LIN {X 0,Y 413.536,Z 977.53,A -85,B 0,C 180,E1 16664.852,E2 16664.852} C_VEL
LIN {X 0,Y 413.201,Z 977.53,A -85,B 0,C 180,E1 16671.503,E2 16671.503} C_VEL
LIN {X 0,Y 412.887,Z 977.53,A -85,B 0,C 180,E1 16678.484,E2 16678.484} C_VEL
LIN {X 0,Y 412.713,Z 977.53,A -85,B 0,C 180,E1 16683.405,E2 16683.405} C_VEL
LIN {X 0,Y 412.557,Z 977.53,A -85,B 0,C 180,E1 16689.514,E2 16689.514} C_VEL
LIN {X 0,Y 412.491,Z 977.53,A -85,B 0,C 180,E1 16695.722,E2 16695.722} C_VEL
LIN {X 0,Y 412.588,Z 977.53,A -85,B 0,C 180,E1 16699.527,E2 16699.527} C_VEL
LIN {X 0,Y 434.551,Z 1034.787,A -85,B 0,C 180,E1 16702.862,E2 16702.862} C_VEL
LIN {X 0,Y 443.784,Z 1065.068,A -85,B 0,C 180,E1 16704.876,E2 16704.876} C_VEL
LIN {X 0,Y 438.617,Z 1105.248,A -85,B 0,C 180,E1 16707.191,E2 16707.191} C_VEL
LIN {X 0,Y 432.749,Z 1141.95,A -85,B 0,C 180,E1 16710.201,E2 16710.201} C_VEL
LIN {X 0,Y 427.169,Z 1174.246,A -85,B 0,C 180,E1 16713.808,E2 16713.808} C_VEL
LIN {X 0,Y 422.467,Z 1201.399,A -85,B 0,C 180,E1 16717.863,E2 16717.863} C_VEL
LIN {X 0,Y 418.685,Z 1224.945,A -85,B 0,C 180,E1 16722.615,E2 16722.615} C_VEL
LIN {X 0,Y 416.229,Z 1243.361,A -85,B 0,C 180,E1 16727.903,E2 16727.903} C_VEL
LIN {X 0,Y 415.214,Z 1254.307,A -85,B 0,C 180,E1 16732.648,E2 16732.648} C_VEL
LIN {X 0,Y 414.843,Z 1260.908,A -85,B 0,C 180,E1 16737.892,E2 16737.892} C_VEL
LIN {X 0,Y 415.006,Z 1262.266,A -85,B 0,C 180,E1 16742.077,E2 16742.077} C_VEL
LIN {X 0,Y 415.617,Z 1259.292,A -85,B 0,C 180,E1 16747.315,E2 16747.315} C_VEL
LIN {X 0,Y 417.308,Z 1251.014,A -85,B 0,C 180,E1 16752.567,E2 16752.567} C_VEL
LIN {X 0,Y 420.683,Z 1237.254,A -85,B 0,C 180,E1 16757.74,E2 16757.74} C_VEL
LIN {X 0,Y 426.06,Z 1217.939,A -85,B 0,C 180,E1 16762.692,E2 16762.692} C_VEL
LIN {X 0,Y 433.442,Z 1192.911,A -85,B 0,C 180,E1 16767.292,E2 16767.292} C_VEL
LIN {X 0,Y 442.539,Z 1161.806,A -85,B 0,C 180,E1 16771.457,E2 16771.457} C_VEL
LIN {X 0,Y 452.529,Z 1126.179,A -85,B 0,C 180,E1 16774.968,E2 16774.968} C_VEL
LIN {X 0,Y 462.553,Z 1087.333,A -85,B 0,C 180,E1 16777.725,E2 16777.725} C_VEL
LIN {X 0,Y 466.359,Z 1070.164,A -85,B 0,C 180,E1 16778.772,E2 16778.772} C_VEL
LIN {X 0,Y 465.511,Z 1057.108,A -85,B 0,C 180,E1 16780.595,E2 16780.595} C_VEL
LIN {X 0,Y 464.2,Z 1049.101,A -85,B 0,C 180,E1 16782.676,E2 16782.676} C_VEL
LIN {X 0,Y 464.109,Z 1045.742,A -85,B 0,C 180,E1 16784.686,E2 16784.686} C_VEL
LIN {X 0,Y 465.124,Z 1051.822,A -85,B 0,C 180,E1 16787.421,E2 16787.421} C_VEL
LIN {X 0,Y 465.932,Z 1056.52,A -85,B 0,C 180,E1 16788.389,E2 16788.389} C_VEL
LIN {X 0,Y 464.634,Z 1082.21,A -85,B 0,C 180,E1 16790.745,E2 16790.745} C_VEL
LIN {X 0,Y 453.94,Z 1125.674,A -85,B 0,C 180,E1 16793.081,E2 16793.081} C_VEL
LIN {X 0,Y 443.218,Z 1167.129,A -85,B 0,C 180,E1 16796.262,E2 16796.262} C_VEL
LIN {X 0,Y 434.228,Z 1201.819,A -85,B 0,C 180,E1 16799.903,E2 16799.903} C_VEL
LIN {X 0,Y 426.431,Z 1232.42,A -85,B 0,C 180,E1 16804.207,E2 16804.207} C_VEL
LIN {X 0,Y 420.735,Z 1257.224,A -85,B 0,C 180,E1 16808.901,E2 16808.901} C_VEL
LIN {X 0,Y 417.082,Z 1276.771,A -85,B 0,C 180,E1 16813.992,E2 16813.992} C_VEL
LIN {X 0,Y 415.427,Z 1289.933,A -85,B 0,C 180,E1 16818.97,E2 16818.97} C_VEL
LIN {X 0,Y 414.983,Z 1297.641,A -85,B 0,C 180,E1 16823.721,E2 16823.721} C_VEL
LIN {X 0,Y 414.942,Z 1300.55,A -85,B 0,C 180,E1 16827.917,E2 16827.917} C_VEL
LIN {X 0,Y 415.003,Z 1299.894,A -85,B 0,C 180,E1 16832.102,E2 16832.102} C_VEL
LIN {X 0,Y 415.091,Z 1293.746,A -85,B 0,C 180,E1 16837.35,E2 16837.35} C_VEL
LIN {X 0,Y 415.76,Z 1281.343,A -85,B 0,C 180,E1 16842.641,E2 16842.641} C_VEL
LIN {X 0,Y 416.754,Z 1270.596,A -85,B 0,C 180,E1 16845.839,E2 16845.839} C_VEL
LIN {X 0,Y 413.815,Z 1262.25,A -85,B 0,C 180,E1 16847.92,E2 16847.92} C_VEL
LIN {X 0,Y 411.157,Z 1253.033,A -85,B 0,C 180,E1 16849.975,E2 16849.975} C_VEL
LIN {X 0,Y 415.427,Z 1226.434,A -85,B 0,C 180,E1 16854.617,E2 16854.617} C_VEL
LIN {X 0,Y 423.644,Z 1186.586,A -85,B 0,C 180,E1 16860.06,E2 16860.06} C_VEL
LIN {X 0,Y 431.531,Z 1151.479,A -85,B 0,C 180,E1 16863.587,E2 16863.587} C_VEL
LIN {X 0,Y 439.938,Z 1112.289,A -85,B 0,C 180,E1 16866.462,E2 16866.462} C_VEL
LIN {X 0,Y 446.354,Z 1076.799,A -85,B 0,C 180,E1 16868.367,E2 16868.367} C_VEL
LIN {X 0,Y 443.694,Z 1053.032,A -85,B 0,C 180,E1 16870.272,E2 16870.272} C_VEL
LIN {X 0,Y 436.241,Z 1030.153,A -85,B 0,C 180,E1 16873.006,E2 16873.006} C_VEL
LIN {X 0,Y 428.199,Z 1013.282,A -85,B 0,C 180,E1 16876.073,E2 16876.073} C_VEL
LIN {X 0,Y 423.144,Z 1004.639,A -85,B 0,C 180,E1 16878.498,E2 16878.498} C_VEL
LIN {X 0,Y 420.285,Z 999.454,A -85,B 0,C 180,E1 16880.39,E2 16880.39} C_VEL
LIN {X 0,Y 416.589,Z 992.929,A -85,B 0,C 180,E1 16886.206,E2 16886.206} C_VEL
LIN {X 0,Y 419.779,Z 999.169,A -85,B 0,C 180,E1 16892.034,E2 16892.034} C_VEL
LIN {X 0,Y 426.481,Z 1011.08,A -85,B 0,C 180,E1 16896.342,E2 16896.342} C_VEL
LIN {X 0,Y 434.002,Z 1026.493,A -85,B 0,C 180,E1 16899.77,E2 16899.77} C_VEL
LIN {X 0,Y 441.381,Z 1046.678,A -85,B 0,C 180,E1 16902.741,E2 16902.741} C_VEL
LIN {X 0,Y 443.164,Z 1055.011,A -85,B 0,C 180,E1 16903.605,E2 16903.605} C_VEL
LIN {X 0,Y 435.927,Z 1100.938,A -85,B 0,C 180,E1 16905.934,E2 16905.934} C_VEL
LIN {X 0,Y 430.586,Z 1128.785,A -85,B 0,C 180,E1 16908.213,E2 16908.213} C_VEL
LIN {X 0,Y 424.859,Z 1152.118,A -85,B 0,C 180,E1 16911.039,E2 16911.039} C_VEL
LIN {X 0,Y 419.666,Z 1170.692,A -85,B 0,C 180,E1 16914.325,E2 16914.325} C_VEL
LIN {X 0,Y 414.89,Z 1185.812,A -85,B 0,C 180,E1 16918.446,E2 16918.446} C_VEL
LIN {X 0,Y 411.879,Z 1193.72,A -85,B 0,C 180,E1 16922.123,E2 16922.123} C_VEL
LIN {X 0,Y 409.732,Z 1197.42,A -85,B 0,C 180,E1 16926.384,E2 16926.384} C_VEL
LIN {X 0,Y 408.96,Z 1195.423,A -85,B 0,C 180,E1 16930.69,E2 16930.69} C_VEL
LIN {X 0,Y 409.267,Z 1187.552,A -85,B 0,C 180,E1 16935.034,E2 16935.034} C_VEL
LIN {X 0,Y 410.416,Z 1173.844,A -85,B 0,C 180,E1 16939.141,E2 16939.141} C_VEL
LIN {X 0,Y 412.34,Z 1154.397,A -85,B 0,C 180,E1 16942.905,E2 16942.905} C_VEL
LIN {X 0,Y 414.797,Z 1130.818,A -85,B 0,C 180,E1 16946.013,E2 16946.013} C_VEL
LIN {X 0,Y 417.4,Z 1103.039,A -85,B 0,C 180,E1 16948.484,E2 16948.484} C_VEL
LIN {X 0,Y 419.403,Z 1073.396,A -85,B 0,C 180,E1 16950.16,E2 16950.16} C_VEL
LIN {X 0,Y 420.294,Z 1032.093,A -85,B 0,C 180,E1 16951.546,E2 16951.546} C_VEL
LIN {X 0,Y 404.933,Z 977.53,A -85,B 0,C 180,E1 16954.16,E2 16954.16} C_VEL
LIN {X 0,Y 404.685,Z 977.53,A -85,B 0,C 180,E1 16961.493,E2 16961.493} C_VEL
LIN {X 0,Y 404.613,Z 977.53,A -85,B 0,C 180,E1 16968.519,E2 16968.519} C_VEL
LIN {X 0,Y 404.669,Z 977.53,A -85,B 0,C 180,E1 16975.817,E2 16975.817} C_VEL
LIN {X 0,Y 404.874,Z 977.53,A -85,B 0,C 180,E1 16980.876,E2 16980.876} C_VEL
LIN {X 0,Y 405.13,Z 977.53,A -85,B 0,C 180,E1 16985.695,E2 16985.695} C_VEL
LIN {X 0,Y 405.516,Z 977.53,A -85,B 0,C 180,E1 16992.596,E2 16992.596} C_VEL
LIN {X 0,Y 405.838,Z 977.53,A -85,B 0,C 180,E1 16999.231,E2 16999.231} C_VEL
LIN {X 0,Y 406.347,Z 977.53,A -85,B 0,C 180,E1 17005.713,E2 17005.713} C_VEL
LIN {X 0,Y 406.535,Z 977.53,A -85,B 0,C 180,E1 17012.126,E2 17012.126} C_VEL
LIN {X 0,Y 405.996,Z 977.53,A -85,B 0,C 180,E1 17018.576,E2 17018.576} C_VEL
LIN {X 0,Y 405.593,Z 977.53,A -85,B 0,C 180,E1 17025.15,E2 17025.15} C_VEL
LIN {X 0,Y 405.24,Z 977.53,A -85,B 0,C 180,E1 17031.947,E2 17031.947} C_VEL
LIN {X 0,Y 404.884,Z 977.53,A -85,B 0,C 180,E1 17039.101,E2 17039.101} C_VEL
LIN {X 0,Y 404.684,Z 977.53,A -85,B 0,C 180,E1 17044.521,E2 17044.521} C_VEL
LIN {X 0,Y 404.658,Z 977.53,A -85,B 0,C 180,E1 17051.488,E2 17051.488} C_VEL
LIN {X 0,Y 404.639,Z 977.53,A -85,B 0,C 180,E1 17058.914,E2 17058.914} C_VEL
LIN {X 0,Y 426.55,Z 1034.457,A -85,B 0,C 180,E1 17062.312,E2 17062.312} C_VEL
LIN {X 0,Y 436.463,Z 1066.891,A -85,B 0,C 180,E1 17064.525,E2 17064.525} C_VEL
LIN {X 0,Y 430.951,Z 1107.765,A -85,B 0,C 180,E1 17066.963,E2 17066.963} C_VEL
LIN {X 0,Y 424.975,Z 1144.124,A -85,B 0,C 180,E1 17070.042,E2 17070.042} C_VEL
LIN {X 0,Y 419.31,Z 1176.038,A -85,B 0,C 180,E1 17073.712,E2 17073.712} C_VEL
LIN {X 0,Y 414.384,Z 1203.666,A -85,B 0,C 180,E1 17077.974,E2 17077.974} C_VEL
LIN {X 0,Y 410.632,Z 1226.719,A -85,B 0,C 180,E1 17082.816,E2 17082.816} C_VEL
LIN {X 0,Y 408.424,Z 1243.246,A -85,B 0,C 180,E1 17087.669,E2 17087.669} C_VEL
LIN {X 0,Y 407.343,Z 1254.386,A -85,B 0,C 180,E1 17092.505,E2 17092.505} C_VEL
LIN {X 0,Y 406.977,Z 1261.213,A -85,B 0,C 180,E1 17097.851,E2 17097.851} C_VEL
LIN {X 0,Y 407.123,Z 1262.708,A -85,B 0,C 180,E1 17102.117,E2 17102.117} C_VEL
LIN {X 0,Y 407.801,Z 1259.921,A -85,B 0,C 180,E1 17107.456,E2 17107.456} C_VEL
LIN {X 0,Y 409.589,Z 1251.856,A -85,B 0,C 180,E1 17112.808,E2 17112.808} C_VEL
LIN {X 0,Y 413.286,Z 1238.13,A -85,B 0,C 180,E1 17118.139,E2 17118.139} C_VEL
LIN {X 0,Y 419.339,Z 1218.042,A -85,B 0,C 180,E1 17123.402,E2 17123.402} C_VEL
LIN {X 0,Y 427.658,Z 1191.664,A -85,B 0,C 180,E1 17128.268,E2 17128.268} C_VEL
LIN {X 0,Y 437.472,Z 1160.499,A -85,B 0,C 180,E1 17132.45,E2 17132.45} C_VEL
LIN {X 0,Y 448.599,Z 1123.62,A -85,B 0,C 180,E1 17136.048,E2 17136.048} C_VEL
LIN {X 0,Y 459.906,Z 1083.35,A -85,B 0,C 180,E1 17138.871,E2 17138.871} C_VEL
LIN {X 0,Y 462.155,Z 1073.258,A -85,B 0,C 180,E1 17139.544,E2 17139.544} C_VEL
LIN {X 0,Y 461.934,Z 1061.361,A -85,B 0,C 180,E1 17141.422,E2 17141.422} C_VEL
LIN {X 0,Y 461.315,Z 1054.684,A -85,B 0,C 180,E1 17143.741,E2 17143.741} C_VEL
LIN {X 0,Y 461.576,Z 1053.795,A -85,B 0,C 180,E1 17145.034,E2 17145.034} C_VEL
LIN {X 0,Y 462.268,Z 1059.274,A -85,B 0,C 180,E1 17147.264,E2 17147.264} C_VEL
LIN {X 0,Y 462.149,Z 1064.747,A -85,B 0,C 180,E1 17148.087,E2 17148.087} C_VEL
LIN {X 0,Y 459.961,Z 1085.959,A -85,B 0,C 180,E1 17150.036,E2 17150.036} C_VEL
LIN {X 0,Y 448.531,Z 1128.125,A -85,B 0,C 180,E1 17152.407,E2 17152.407} C_VEL
LIN {X 0,Y 436.938,Z 1169.453,A -85,B 0,C 180,E1 17155.711,E2 17155.711} C_VEL
LIN {X 0,Y 426.936,Z 1205.032,A -85,B 0,C 180,E1 17159.63,E2 17159.63} C_VEL
LIN {X 0,Y 418.917,Z 1234.622,A -85,B 0,C 180,E1 17163.998,E2 17163.998} C_VEL
LIN {X 0,Y 412.8,Z 1259.522,A -85,B 0,C 180,E1 17168.96,E2 17168.96} C_VEL
LIN {X 0,Y 409.067,Z 1278.74,A -85,B 0,C 180,E1 17174.304,E2 17174.304} C_VEL
LIN {X 0,Y 407.475,Z 1290.882,A -85,B 0,C 180,E1 17179.295,E2 17179.295} C_VEL
LIN {X 0,Y 407.093,Z 1297.34,A -85,B 0,C 180,E1 17183.599,E2 17183.599} C_VEL
LIN {X 0,Y 407.054,Z 1300.164,A -85,B 0,C 180,E1 17187.877,E2 17187.877} C_VEL
LIN {X 0,Y 407.111,Z 1299.389,A -85,B 0,C 180,E1 17192.143,E2 17192.143} C_VEL
LIN {X 0,Y 407.151,Z 1294.742,A -85,B 0,C 180,E1 17196.42,E2 17196.42} C_VEL
LIN {X 0,Y 407.568,Z 1284.889,A -85,B 0,C 180,E1 17201.266,E2 17201.266} C_VEL
LIN {X 0,Y 409.036,Z 1268.898,A -85,B 0,C 180,E1 17206.306,E2 17206.306} C_VEL
LIN {X 0,Y 411.157,Z 1253.033,A -85,B 0,C 180,E1 17209.975,E2 17209.975} C_VEL
LIN {X 0,Y 408.709,Z 1243.141,A -85,B 0,C 180,E1 17211.973,E2 17211.973} C_VEL
LIN {X 0,Y 406.726,Z 1232.323,A -85,B 0,C 180,E1 17213.894,E2 17213.894} C_VEL
LIN {X 0,Y 414.524,Z 1196.057,A -85,B 0,C 180,E1 17219.43,E2 17219.43} C_VEL
LIN {X 0,Y 422.708,Z 1161.586,A -85,B 0,C 180,E1 17223.303,E2 17223.303} C_VEL
LIN {X 0,Y 431.811,Z 1122.039,A -85,B 0,C 180,E1 17226.533,E2 17226.533} C_VEL
LIN {X 0,Y 440.546,Z 1079.46,A -85,B 0,C 180,E1 17228.968,E2 17228.968} C_VEL
LIN {X 0,Y 438.447,Z 1056.769,A -85,B 0,C 180,E1 17230.875,E2 17230.875} C_VEL
LIN {X 0,Y 431.79,Z 1034.922,A -85,B 0,C 180,E1 17233.622,E2 17233.622} C_VEL
LIN {X 0,Y 424.344,Z 1018.331,A -85,B 0,C 180,E1 17236.819,E2 17236.819} C_VEL
LIN {X 0,Y 418.261,Z 1007.062,A -85,B 0,C 180,E1 17240.432,E2 17240.432} C_VEL
LIN {X 0,Y 414.556,Z 1000.548,A -85,B 0,C 180,E1 17246.035,E2 17246.035} C_VEL
LIN {X 0,Y 415.519,Z 1004.822,A -85,B 0,C 180,E1 17250.297,E2 17250.297} C_VEL
LIN {X 0,Y 417.924,Z 1008.082,A -85,B 0,C 180,E1 17252.561,E2 17252.561} C_VEL
LIN {X 0,Y 424.057,Z 1019.723,A -85,B 0,C 180,E1 17256.566,E2 17256.566} C_VEL
LIN {X 0,Y 431.211,Z 1036.04,A -85,B 0,C 180,E1 17260.013,E2 17260.013} C_VEL
LIN {X 0,Y 437.52,Z 1056.068,A -85,B 0,C 180,E1 17262.818,E2 17262.818} C_VEL
LIN {X 0,Y 429.787,Z 1103.231,A -85,B 0,C 180,E1 17265.338,E2 17265.338} C_VEL
LIN {X 0,Y 424.151,Z 1130.371,A -85,B 0,C 180,E1 17267.639,E2 17267.639} C_VEL
LIN {X 0,Y 417.897,Z 1154.294,A -85,B 0,C 180,E1 17270.625,E2 17270.625} C_VEL
LIN {X 0,Y 412.226,Z 1173.211,A -85,B 0,C 180,E1 17274.129,E2 17274.129} C_VEL
LIN {X 0,Y 407.693,Z 1186.506,A -85,B 0,C 180,E1 17277.885,E2 17277.885} C_VEL
LIN {X 0,Y 404.055,Z 1195.396,A -85,B 0,C 180,E1 17282.164,E2 17282.164} C_VEL
LIN {X 0,Y 401.849,Z 1198.507,A -85,B 0,C 180,E1 17286.51,E2 17286.51} C_VEL
LIN {X 0,Y 401.121,Z 1196.049,A -85,B 0,C 180,E1 17290.902,E2 17290.902} C_VEL
LIN {X 0,Y 401.451,Z 1187.613,A -85,B 0,C 180,E1 17295.334,E2 17295.334} C_VEL
LIN {X 0,Y 402.68,Z 1173.379,A -85,B 0,C 180,E1 17299.523,E2 17299.523} C_VEL
LIN {X 0,Y 404.655,Z 1153.91,A -85,B 0,C 180,E1 17303.244,E2 17303.244} C_VEL
LIN {X 0,Y 407.234,Z 1129.906,A -85,B 0,C 180,E1 17306.384,E2 17306.384} C_VEL
LIN {X 0,Y 409.884,Z 1102.27,A -85,B 0,C 180,E1 17308.834,E2 17308.834} C_VEL
LIN {X 0,Y 411.856,Z 1071.439,A -85,B 0,C 180,E1 17310.558,E2 17310.558} C_VEL
LIN {X 0,Y 412.97,Z 1034.333,A -85,B 0,C 180,E1 17311.814,E2 17311.814} C_VEL
LIN {X 0,Y 396.984,Z 977.53,A -85,B 0,C 180,E1 17314.608,E2 17314.608} C_VEL
LIN {X 0,Y 396.738,Z 977.53,A -85,B 0,C 180,E1 17320.502,E2 17320.502} C_VEL
LIN {X 0,Y 396.628,Z 977.53,A -85,B 0,C 180,E1 17326.557,E2 17326.557} C_VEL
LIN {X 0,Y 396.697,Z 977.53,A -85,B 0,C 180,E1 17333.352,E2 17333.352} C_VEL
LIN {X 0,Y 396.933,Z 977.53,A -85,B 0,C 180,E1 17340.235,E2 17340.235} C_VEL
LIN {X 0,Y 397.284,Z 977.53,A -85,B 0,C 180,E1 17347.568,E2 17347.568} C_VEL
LIN {X 0,Y 397.651,Z 977.53,A -85,B 0,C 180,E1 17354.519,E2 17354.519} C_VEL
LIN {X 0,Y 398.124,Z 977.53,A -85,B 0,C 180,E1 17361.776,E2 17361.776} C_VEL
LIN {X 0,Y 398.591,Z 977.53,A -85,B 0,C 180,E1 17367.811,E2 17367.811} C_VEL
LIN {X 0,Y 398.623,Z 977.53,A -85,B 0,C 180,E1 17372.168,E2 17372.168} C_VEL
LIN {X 0,Y 398.066,Z 977.53,A -85,B 0,C 180,E1 17378.748,E2 17378.748} C_VEL
LIN {X 0,Y 397.64,Z 977.53,A -85,B 0,C 180,E1 17385.46,E2 17385.46} C_VEL
LIN {X 0,Y 397.255,Z 977.53,A -85,B 0,C 180,E1 17392.411,E2 17392.411} C_VEL
LIN {X 0,Y 396.938,Z 977.53,A -85,B 0,C 180,E1 17399.741,E2 17399.741} C_VEL
LIN {X 0,Y 396.726,Z 977.53,A -85,B 0,C 180,E1 17406.654,E2 17406.654} C_VEL
LIN {X 0,Y 396.66,Z 977.53,A -85,B 0,C 180,E1 17413.448,E2 17413.448} C_VEL
LIN {X 0,Y 396.705,Z 977.53,A -85,B 0,C 180,E1 17418.264,E2 17418.264} C_VEL
LIN {X 0,Y 419.101,Z 1035.699,A -85,B 0,C 180,E1 17421.852,E2 17421.852} C_VEL
LIN {X 0,Y 429.116,Z 1068.588,A -85,B 0,C 180,E1 17424.155,E2 17424.155} C_VEL
LIN {X 0,Y 423.515,Z 1108.732,A -85,B 0,C 180,E1 17426.614,E2 17426.614} C_VEL
LIN {X 0,Y 417.45,Z 1144.782,A -85,B 0,C 180,E1 17429.726,E2 17429.726} C_VEL
LIN {X 0,Y 411.631,Z 1176.792,A -85,B 0,C 180,E1 17433.478,E2 17433.478} C_VEL
LIN {X 0,Y 406.586,Z 1204.37,A -85,B 0,C 180,E1 17437.817,E2 17437.817} C_VEL
LIN {X 0,Y 402.761,Z 1227.315,A -85,B 0,C 180,E1 17442.742,E2 17442.742} C_VEL
LIN {X 0,Y 400.434,Z 1244.556,A -85,B 0,C 180,E1 17447.973,E2 17447.973} C_VEL
LIN {X 0,Y 399.488,Z 1254.42,A -85,B 0,C 180,E1 17452.356,E2 17452.356} C_VEL
LIN {X 0,Y 399.078,Z 1261.475,A -85,B 0,C 180,E1 17457.809,E2 17457.809} C_VEL
LIN {X 0,Y 399.234,Z 1263.156,A -85,B 0,C 180,E1 17462.159,E2 17462.159} C_VEL
LIN {X 0,Y 399.974,Z 1260.569,A -85,B 0,C 180,E1 17467.603,E2 17467.603} C_VEL
LIN {X 0,Y 401.881,Z 1252.733,A -85,B 0,C 180,E1 17473.058,E2 17473.058} C_VEL
LIN {X 0,Y 405.841,Z 1239.276,A -85,B 0,C 180,E1 17478.485,E2 17478.485} C_VEL
LIN {X 0,Y 412.219,Z 1219.565,A -85,B 0,C 180,E1 17483.831,E2 17483.831} C_VEL
LIN {X 0,Y 420.995,Z 1193.848,A -85,B 0,C 180,E1 17488.756,E2 17488.756} C_VEL
LIN {X 0,Y 431.625,Z 1162.505,A -85,B 0,C 180,E1 17493.095,E2 17493.095} C_VEL
LIN {X 0,Y 443.394,Z 1126.739,A -85,B 0,C 180,E1 17496.708,E2 17496.708} C_VEL
LIN {X 0,Y 455.543,Z 1087.183,A -85,B 0,C 180,E1 17499.59,E2 17499.59} C_VEL
LIN {X 0,Y 458.267,Z 1076.739,A -85,B 0,C 180,E1 17500.305,E2 17500.305} C_VEL
LIN {X 0,Y 458.594,Z 1066.761,A -85,B 0,C 180,E1 17502.065,E2 17502.065} C_VEL
LIN {X 0,Y 458.613,Z 1061.998,A -85,B 0,C 180,E1 17503.91,E2 17503.91} C_VEL
LIN {X 0,Y 458.836,Z 1061.482,A -85,B 0,C 180,E1 17505.063,E2 17505.063} C_VEL
LIN {X 0,Y 459.199,Z 1065.972,A -85,B 0,C 180,E1 17506.909,E2 17506.909} C_VEL
LIN {X 0,Y 456.734,Z 1084.393,A -85,B 0,C 180,E1 17508.934,E2 17508.934} C_VEL
LIN {X 0,Y 441.705,Z 1136.16,A -85,B 0,C 180,E1 17512.106,E2 17512.106} C_VEL
LIN {X 0,Y 429.188,Z 1176.718,A -85,B 0,C 180,E1 17515.617,E2 17515.617} C_VEL
LIN {X 0,Y 418.299,Z 1212.873,A -85,B 0,C 180,E1 17519.97,E2 17519.97} C_VEL
LIN {X 0,Y 410.135,Z 1241.628,A -85,B 0,C 180,E1 17524.676,E2 17524.676} C_VEL
LIN {X 0,Y 404.633,Z 1263.027,A -85,B 0,C 180,E1 17529.361,E2 17529.361} C_VEL
LIN {X 0,Y 400.982,Z 1280.599,A -85,B 0,C 180,E1 17534.672,E2 17534.672} C_VEL
LIN {X 0,Y 399.507,Z 1292.048,A -85,B 0,C 180,E1 17539.837,E2 17539.837} C_VEL
LIN {X 0,Y 399.195,Z 1297.048,A -85,B 0,C 180,E1 17543.472,E2 17543.472} C_VEL
LIN {X 0,Y 399.156,Z 1299.775,A -85,B 0,C 180,E1 17547.835,E2 17547.835} C_VEL
LIN {X 0,Y 399.22,Z 1298.841,A -85,B 0,C 180,E1 17552.185,E2 17552.185} C_VEL
LIN {X 0,Y 399.264,Z 1294.081,A -85,B 0,C 180,E1 17556.548,E2 17556.548} C_VEL
LIN {X 0,Y 399.715,Z 1284.023,A -85,B 0,C 180,E1 17561.49,E2 17561.49} C_VEL
LIN {X 0,Y 401.192,Z 1268.398,A -85,B 0,C 180,E1 17566.466,E2 17566.466} C_VEL
LIN {X 0,Y 404.142,Z 1247.252,A -85,B 0,C 180,E1 17571.248,E2 17571.248} C_VEL
LIN {X 0,Y 406.726,Z 1232.323,A -85,B 0,C 180,E1 17573.894,E2 17573.894} C_VEL
LIN {X 0,Y 405.15,Z 1221.758,A -85,B 0,C 180,E1 17575.852,E2 17575.852} C_VEL
LIN {X 0,Y 403.783,Z 1211.089,A -85,B 0,C 180,E1 17577.819,E2 17577.819} C_VEL
LIN {X 0,Y 411.821,Z 1179.033,A -85,B 0,C 180,E1 17582.112,E2 17582.112} C_VEL
LIN {X 0,Y 421.33,Z 1141.248,A -85,B 0,C 180,E1 17585.793,E2 17585.793} C_VEL
LIN {X 0,Y 430.998,Z 1100.356,A -85,B 0,C 180,E1 17588.624,E2 17588.624} C_VEL
LIN {X 0,Y 434.777,Z 1080.838,A -85,B 0,C 180,E1 17589.697,E2 17589.697} C_VEL
LIN {X 0,Y 433.109,Z 1059.718,A -85,B 0,C 180,E1 17591.582,E2 17591.582} C_VEL
LIN {X 0,Y 426.991,Z 1038.703,A -85,B 0,C 180,E1 17594.426,E2 17594.426} C_VEL
LIN {X 0,Y 420.286,Z 1023.051,A -85,B 0,C 180,E1 17597.698,E2 17597.698} C_VEL
LIN {X 0,Y 415.391,Z 1014.15,A -85,B 0,C 180,E1 17600.949,E2 17600.949} C_VEL
LIN {X 0,Y 412.407,Z 1008.203,A -85,B 0,C 180,E1 17605.695,E2 17605.695} C_VEL
LIN {X 0,Y 412.319,Z 1010.467,A -85,B 0,C 180,E1 17608.7,E2 17608.7} C_VEL
LIN {X 0,Y 415.089,Z 1015.364,A -85,B 0,C 180,E1 17612.357,E2 17612.357} C_VEL
LIN {X 0,Y 420.765,Z 1026.999,A -85,B 0,C 180,E1 17616.403,E2 17616.403} C_VEL
LIN {X 0,Y 427.441,Z 1043.484,A -85,B 0,C 180,E1 17619.884,E2 17619.884} C_VEL
LIN {X 0,Y 432.021,Z 1060.552,A -85,B 0,C 180,E1 17622.244,E2 17622.244} C_VEL
LIN {X 0,Y 424.074,Z 1103.904,A -85,B 0,C 180,E1 17624.605,E2 17624.605} C_VEL
LIN {X 0,Y 417.817,Z 1132.19,A -85,B 0,C 180,E1 17627.049,E2 17627.049} C_VEL
LIN {X 0,Y 410.962,Z 1156.535,A -85,B 0,C 180,E1 17630.198,E2 17630.198} C_VEL
LIN {X 0,Y 405.257,Z 1174.219,A -85,B 0,C 180,E1 17633.576,E2 17633.576} C_VEL
LIN {X 0,Y 399.957,Z 1188.755,A -85,B 0,C 180,E1 17637.845,E2 17637.845} C_VEL
LIN {X 0,Y 396.233,Z 1196.962,A -85,B 0,C 180,E1 17642.207,E2 17642.207} C_VEL
LIN {X 0,Y 393.97,Z 1199.598,A -85,B 0,C 180,E1 17646.641,E2 17646.641} C_VEL
LIN {X 0,Y 393.258,Z 1196.591,A -85,B 0,C 180,E1 17651.123,E2 17651.123} C_VEL
LIN {X 0,Y 393.685,Z 1187.339,A -85,B 0,C 180,E1 17655.76,E2 17655.76} C_VEL
LIN {X 0,Y 395.011,Z 1172.824,A -85,B 0,C 180,E1 17659.906,E2 17659.906} C_VEL
LIN {X 0,Y 397.105,Z 1153.015,A -85,B 0,C 180,E1 17663.657,E2 17663.657} C_VEL
LIN {X 0,Y 399.795,Z 1127.631,A -85,B 0,C 180,E1 17666.914,E2 17666.914} C_VEL
LIN {X 0,Y 402.455,Z 1099.688,A -85,B 0,C 180,E1 17669.319,E2 17669.319} C_VEL
LIN {X 0,Y 404.451,Z 1068.492,A -85,B 0,C 180,E1 17670.995,E2 17670.995} C_VEL
LIN {X 0,Y 405.272,Z 1035.045,A -85,B 0,C 180,E1 17672.148,E2 17672.148} C_VEL
LIN {X 0,Y 389.001,Z 977.53,A -85,B 0,C 180,E1 17675.096,E2 17675.096} C_VEL
LIN {X 0,Y 388.68,Z 977.53,A -85,B 0,C 180,E1 17682.193,E2 17682.193} C_VEL
LIN {X 0,Y 388.635,Z 977.53,A -85,B 0,C 180,E1 17688.471,E2 17688.471} C_VEL
LIN {X 0,Y 388.8,Z 977.53,A -85,B 0,C 180,E1 17694.946,E2 17694.946} C_VEL
LIN {X 0,Y 389.054,Z 977.53,A -85,B 0,C 180,E1 17702.125,E2 17702.125} C_VEL
LIN {X 0,Y 389.463,Z 977.53,A -85,B 0,C 180,E1 17709.492,E2 17709.492} C_VEL
LIN {X 0,Y 389.851,Z 977.53,A -85,B 0,C 180,E1 17716.503,E2 17716.503} C_VEL
LIN {X 0,Y 390.369,Z 977.53,A -85,B 0,C 180,E1 17723.302,E2 17723.302} C_VEL
LIN {X 0,Y 390.881,Z 977.53,A -85,B 0,C 180,E1 17729.99,E2 17729.99} C_VEL
LIN {X 0,Y 390.332,Z 977.53,A -85,B 0,C 180,E1 17736.677,E2 17736.677} C_VEL
LIN {X 0,Y 389.838,Z 977.53,A -85,B 0,C 180,E1 17743.617,E2 17743.617} C_VEL
LIN {X 0,Y 389.406,Z 977.53,A -85,B 0,C 180,E1 17750.923,E2 17750.923} C_VEL
LIN {X 0,Y 389.054,Z 977.53,A -85,B 0,C 180,E1 17757.852,E2 17757.852} C_VEL
LIN {X 0,Y 388.864,Z 977.53,A -85,B 0,C 180,E1 17765.068,E2 17765.068} C_VEL
LIN {X 0,Y 388.687,Z 977.53,A -85,B 0,C 180,E1 17772.193,E2 17772.193} C_VEL
LIN {X 0,Y 388.845,Z 978.262,A -85,B 0,C 180,E1 17777.674,E2 17777.674} C_VEL
LIN {X 0,Y 410.325,Z 1033.448,A -85,B 0,C 180,E1 17781.138,E2 17781.138} C_VEL
LIN {X 0,Y 421.734,Z 1070.249,A -85,B 0,C 180,E1 17783.782,E2 17783.782} C_VEL
LIN {X 0,Y 416.111,Z 1109.544,A -85,B 0,C 180,E1 17786.253,E2 17786.253} C_VEL
LIN {X 0,Y 409.883,Z 1145.668,A -85,B 0,C 180,E1 17789.435,E2 17789.435} C_VEL
LIN {X 0,Y 403.97,Z 1177.456,A -85,B 0,C 180,E1 17793.235,E2 17793.235} C_VEL
LIN {X 0,Y 398.788,Z 1205.002,A -85,B 0,C 180,E1 17797.654,E2 17797.654} C_VEL
LIN {X 0,Y 394.922,Z 1227.672,A -85,B 0,C 180,E1 17802.613,E2 17802.613} C_VEL
LIN {X 0,Y 392.609,Z 1244.393,A -85,B 0,C 180,E1 17807.73,E2 17807.73} C_VEL
LIN {X 0,Y 391.618,Z 1254.437,A -85,B 0,C 180,E1 17812.202,E2 17812.202} C_VEL
LIN {X 0,Y 391.189,Z 1261.717,A -85,B 0,C 180,E1 17817.765,E2 17817.765} C_VEL
LIN {X 0,Y 391.361,Z 1263.605,A -85,B 0,C 180,E1 17822.203,E2 17822.203} C_VEL
LIN {X 0,Y 391.867,Z 1262.108,A -85,B 0,C 180,E1 17826.645,E2 17826.645} C_VEL
LIN {X 0,Y 393.671,Z 1255.563,A -85,B 0,C 180,E1 17832.204,E2 17832.204} C_VEL
LIN {X 0,Y 397.312,Z 1243.592,A -85,B 0,C 180,E1 17837.746,E2 17837.746} C_VEL
LIN {X 0,Y 403.819,Z 1224.829,A -85,B 0,C 180,E1 17843.408,E2 17843.408} C_VEL
LIN {X 0,Y 412.763,Z 1200.513,A -85,B 0,C 180,E1 17848.484,E2 17848.484} C_VEL
LIN {X 0,Y 423.128,Z 1172.44,A -85,B 0,C 180,E1 17852.774,E2 17852.774} C_VEL
LIN {X 0,Y 435.535,Z 1137.932,A -85,B 0,C 180,E1 17856.66,E2 17856.66} C_VEL
LIN {X 0,Y 449.097,Z 1098.521,A -85,B 0,C 180,E1 17859.848,E2 17859.848} C_VEL
LIN {X 0,Y 454.543,Z 1081.55,A -85,B 0,C 180,E1 17860.939,E2 17860.939} C_VEL
LIN {X 0,Y 455.425,Z 1073.391,A -85,B 0,C 180,E1 17862.426,E2 17862.426} C_VEL
LIN {X 0,Y 455.796,Z 1069.201,A -85,B 0,C 180,E1 17864.252,E2 17864.252} C_VEL
LIN {X 0,Y 456.008,Z 1071.424,A -85,B 0,C 180,E1 17866.175,E2 17866.175} C_VEL
LIN {X 0,Y 455.611,Z 1074.544,A -85,B 0,C 180,E1 17866.763,E2 17866.763} C_VEL
LIN {X 0,Y 452.214,Z 1091.112,A -85,B 0,C 180,E1 17868.416,E2 17868.416} C_VEL
LIN {X 0,Y 438.117,Z 1134.084,A -85,B 0,C 180,E1 17871.033,E2 17871.033} C_VEL
LIN {X 0,Y 424.153,Z 1175.777,A -85,B 0,C 180,E1 17874.681,E2 17874.681} C_VEL
LIN {X 0,Y 412.454,Z 1211.637,A -85,B 0,C 180,E1 17879.059,E2 17879.059} C_VEL
LIN {X 0,Y 403.687,Z 1239.752,A -85,B 0,C 180,E1 17883.685,E2 17883.685} C_VEL
LIN {X 0,Y 397.393,Z 1262.1,A -85,B 0,C 180,E1 17888.626,E2 17888.626} C_VEL
LIN {X 0,Y 393.521,Z 1279.282,A -85,B 0,C 180,E1 17893.858,E2 17893.858} C_VEL
LIN {X 0,Y 391.645,Z 1291.668,A -85,B 0,C 180,E1 17899.504,E2 17899.504} C_VEL
LIN {X 0,Y 391.315,Z 1296.763,A -85,B 0,C 180,E1 17903.339,E2 17903.339} C_VEL
LIN {X 0,Y 391.258,Z 1299.389,A -85,B 0,C 180,E1 17907.791,E2 17907.791} C_VEL
LIN {X 0,Y 391.357,Z 1298.286,A -85,B 0,C 180,E1 17912.229,E2 17912.229} C_VEL
LIN {X 0,Y 391.381,Z 1293.402,A -85,B 0,C 180,E1 17916.68,E2 17916.68} C_VEL
LIN {X 0,Y 391.895,Z 1283.119,A -85,B 0,C 180,E1 17921.722,E2 17921.722} C_VEL
LIN {X 0,Y 393.456,Z 1267.225,A -85,B 0,C 180,E1 17926.799,E2 17926.799} C_VEL
LIN {X 0,Y 396.471,Z 1246.163,A -85,B 0,C 180,E1 17931.594,E2 17931.594} C_VEL
LIN {X 0,Y 403.783,Z 1211.089,A -85,B 0,C 180,E1 17937.819,E2 17937.819} C_VEL
LIN {X 0,Y 402.993,Z 1200.026,A -85,B 0,C 180,E1 17939.749,E2 17939.749} C_VEL
LIN {X 0,Y 402.754,Z 1188.376,A -85,B 0,C 180,E1 17941.614,E2 17941.614} C_VEL
LIN {X 0,Y 412.441,Z 1152.501,A -85,B 0,C 180,E1 17945.528,E2 17945.528} C_VEL
LIN {X 0,Y 422.357,Z 1113.696,A -85,B 0,C 180,E1 17948.573,E2 17948.573} C_VEL
LIN {X 0,Y 429.164,Z 1082.342,A -85,B 0,C 180,E1 17950.447,E2 17950.447} C_VEL
LIN {X 0,Y 428.047,Z 1063.831,A -85,B 0,C 180,E1 17952.178,E2 17952.178} C_VEL
LIN {X 0,Y 422.672,Z 1043.689,A -85,B 0,C 180,E1 17955.047,E2 17955.047} C_VEL
LIN {X 0,Y 416.915,Z 1029.278,A -85,B 0,C 180,E1 17958.23,E2 17958.23} C_VEL
LIN {X 0,Y 412.722,Z 1021.415,A -85,B 0,C 180,E1 17961.25,E2 17961.25} C_VEL
LIN {X 0,Y 410.04,Z 1015.71,A -85,B 0,C 180,E1 17966.359,E2 17966.359} C_VEL
LIN {X 0,Y 412.069,Z 1022.185,A -85,B 0,C 180,E1 17971.97,E2 17971.97} C_VEL
LIN {X 0,Y 416.807,Z 1032.693,A -85,B 0,C 180,E1 17975.828,E2 17975.828} C_VEL
LIN {X 0,Y 422.958,Z 1049.005,A -85,B 0,C 180,E1 17979.421,E2 17979.421} C_VEL
LIN {X 0,Y 426.643,Z 1063.348,A -85,B 0,C 180,E1 17981.529,E2 17981.529} C_VEL
LIN {X 0,Y 418.201,Z 1106.168,A -85,B 0,C 180,E1 17983.95,E2 17983.95} C_VEL
LIN {X 0,Y 411.522,Z 1134.031,A -85,B 0,C 180,E1 17986.441,E2 17986.441} C_VEL
LIN {X 0,Y 404.629,Z 1157.175,A -85,B 0,C 180,E1 17989.498,E2 17989.498} C_VEL
LIN {X 0,Y 398.1,Z 1176.08,A -85,B 0,C 180,E1 17993.185,E2 17993.185} C_VEL
LIN {X 0,Y 392.821,Z 1189.539,A -85,B 0,C 180,E1 17997.252,E2 17997.252} C_VEL
LIN {X 0,Y 389.178,Z 1197.16,A -85,B 0,C 180,E1 18001.131,E2 18001.131} C_VEL
LIN {X 0,Y 387.069,Z 1200.283,A -85,B 0,C 180,E1 18004.506,E2 18004.506} C_VEL
LIN {X 0,Y 385.552,Z 1199.561,A -85,B 0,C 180,E1 18009.06,E2 18009.06} C_VEL
LIN {X 0,Y 385.504,Z 1193.161,A -85,B 0,C 180,E1 18013.656,E2 18013.656} C_VEL
LIN {X 0,Y 386.353,Z 1181.233,A -85,B 0,C 180,E1 18018.005,E2 18018.005} C_VEL
LIN {X 0,Y 388.138,Z 1163.661,A -85,B 0,C 180,E1 18022.085,E2 18022.085} C_VEL
LIN {X 0,Y 390.711,Z 1141.76,A -85,B 0,C 180,E1 18025.533,E2 18025.533} C_VEL
LIN {X 0,Y 393.333,Z 1116.179,A -85,B 0,C 180,E1 18028.329,E2 18028.329} C_VEL
LIN {X 0,Y 395.858,Z 1087.075,A -85,B 0,C 180,E1 18030.427,E2 18030.427} C_VEL
LIN {X 0,Y 397.658,Z 1052.431,A -85,B 0,C 180,E1 18031.887,E2 18031.887} C_VEL
LIN {X 0,Y 397.638,Z 1036.142,A -85,B 0,C 180,E1 18032.473,E2 18032.473} C_VEL
LIN {X 0,Y 381.039,Z 977.53,A -85,B 0,C 180,E1 18035.537,E2 18035.537} C_VEL
LIN {X 0,Y 380.724,Z 977.53,A -85,B 0,C 180,E1 18042.594,E2 18042.594} C_VEL
LIN {X 0,Y 380.661,Z 977.53,A -85,B 0,C 180,E1 18049.157,E2 18049.157} C_VEL
LIN {X 0,Y 380.921,Z 977.53,A -85,B 0,C 180,E1 18056.672,E2 18056.672} C_VEL
LIN {X 0,Y 381.235,Z 977.53,A -85,B 0,C 180,E1 18064.062,E2 18064.062} C_VEL
LIN {X 0,Y 381.627,Z 977.53,A -85,B 0,C 180,E1 18071.468,E2 18071.468} C_VEL
LIN {X 0,Y 382.037,Z 977.53,A -85,B 0,C 180,E1 18078.551,E2 18078.551} C_VEL
LIN {X 0,Y 382.614,Z 977.53,A -85,B 0,C 180,E1 18085.447,E2 18085.447} C_VEL
LIN {X 0,Y 382.978,Z 977.53,A -85,B 0,C 180,E1 18089.989,E2 18089.989} C_VEL
LIN {X 0,Y 382.399,Z 977.53,A -85,B 0,C 180,E1 18096.817,E2 18096.817} C_VEL
LIN {X 0,Y 381.93,Z 977.53,A -85,B 0,C 180,E1 18103.76,E2 18103.76} C_VEL
LIN {X 0,Y 381.517,Z 977.53,A -85,B 0,C 180,E1 18110.932,E2 18110.932} C_VEL
LIN {X 0,Y 381.05,Z 977.53,A -85,B 0,C 180,E1 18118.49,E2 18118.49} C_VEL
LIN {X 0,Y 380.941,Z 977.53,A -85,B 0,C 180,E1 18123.827,E2 18123.827} C_VEL
LIN {X 0,Y 380.733,Z 977.53,A -85,B 0,C 180,E1 18130.855,E2 18130.855} C_VEL
LIN {X 0,Y 380.866,Z 977.913,A -85,B 0,C 180,E1 18136.982,E2 18136.982} C_VEL
LIN {X 0,Y 402.828,Z 1034.577,A -85,B 0,C 180,E1 18140.648,E2 18140.648} C_VEL
LIN {X 0,Y 414.384,Z 1071.969,A -85,B 0,C 180,E1 18143.411,E2 18143.411} C_VEL
LIN {X 0,Y 408.408,Z 1112.007,A -85,B 0,C 180,E1 18146.01,E2 18146.01} C_VEL
LIN {X 0,Y 401.918,Z 1148.964,A -85,B 0,C 180,E1 18149.392,E2 18149.392} C_VEL
LIN {X 0,Y 395.71,Z 1181.37,A -85,B 0,C 180,E1 18153.453,E2 18153.453} C_VEL
LIN {X 0,Y 390.408,Z 1208.841,A -85,B 0,C 180,E1 18158.129,E2 18158.129} C_VEL
LIN {X 0,Y 386.848,Z 1229.558,A -85,B 0,C 180,E1 18162.901,E2 18162.901} C_VEL
LIN {X 0,Y 384.62,Z 1245.661,A -85,B 0,C 180,E1 18168.048,E2 18168.048} C_VEL
LIN {X 0,Y 383.546,Z 1256.406,A -85,B 0,C 180,E1 18173.178,E2 18173.178} C_VEL
LIN {X 0,Y 383.291,Z 1261.949,A -85,B 0,C 180,E1 18177.718,E2 18177.718} C_VEL
LIN {X 0,Y 383.473,Z 1264.057,A -85,B 0,C 180,E1 18182.248,E2 18182.248} C_VEL
LIN {X 0,Y 384.04,Z 1262.716,A -85,B 0,C 180,E1 18186.781,E2 18186.781} C_VEL
LIN {X 0,Y 385.947,Z 1256.423,A -85,B 0,C 180,E1 18192.452,E2 18192.452} C_VEL
LIN {X 0,Y 389.85,Z 1244.753,A -85,B 0,C 180,E1 18198.097,E2 18198.097} C_VEL
LIN {X 0,Y 396.684,Z 1226.571,A -85,B 0,C 180,E1 18203.813,E2 18203.813} C_VEL
LIN {X 0,Y 406.129,Z 1202.786,A -85,B 0,C 180,E1 18208.993,E2 18208.993} C_VEL
LIN {X 0,Y 417.564,Z 1174.131,A -85,B 0,C 180,E1 18213.515,E2 18213.515} C_VEL
LIN {X 0,Y 431.217,Z 1139.264,A -85,B 0,C 180,E1 18217.538,E2 18217.538} C_VEL
LIN {X 0,Y 445.487,Z 1101.494,A -85,B 0,C 180,E1 18220.664,E2 18220.664} C_VEL
LIN {X 0,Y 451.252,Z 1085.433,A -85,B 0,C 180,E1 18221.735,E2 18221.735} C_VEL
LIN {X 0,Y 452.462,Z 1078.353,A -85,B 0,C 180,E1 18223.33,E2 18223.33} C_VEL
LIN {X 0,Y 452.802,Z 1076.825,A -85,B 0,C 180,E1 18224.622,E2 18224.622} C_VEL
LIN {X 0,Y 452.95,Z 1078.428,A -85,B 0,C 180,E1 18225.918,E2 18225.918} C_VEL
LIN {X 0,Y 448.965,Z 1093.664,A -85,B 0,C 180,E1 18227.558,E2 18227.558} C_VEL
LIN {X 0,Y 433.698,Z 1135.792,A -85,B 0,C 180,E1 18230.201,E2 18230.201} C_VEL
LIN {X 0,Y 418.494,Z 1177.466,A -85,B 0,C 180,E1 18233.97,E2 18233.97} C_VEL
LIN {X 0,Y 405.842,Z 1213.176,A -85,B 0,C 180,E1 18238.498,E2 18238.498} C_VEL
LIN {X 0,Y 396.723,Z 1240.263,A -85,B 0,C 180,E1 18243.112,E2 18243.112} C_VEL
LIN {X 0,Y 389.898,Z 1262.72,A -85,B 0,C 180,E1 18248.256,E2 18248.256} C_VEL
LIN {X 0,Y 385.525,Z 1280.709,A -85,B 0,C 180,E1 18254.041,E2 18254.041} C_VEL
LIN {X 0,Y 383.704,Z 1292.487,A -85,B 0,C 180,E1 18259.889,E2 18259.889} C_VEL
LIN {X 0,Y 383.34,Z 1298.189,A -85,B 0,C 180,E1 18265.476,E2 18265.476} C_VEL
LIN {X 0,Y 383.586,Z 1298.844,A -85,B 0,C 180,E1 18270.011,E2 18270.011} C_VEL
LIN {X 0,Y 383.537,Z 1294.336,A -85,B 0,C 180,E1 18275.679,E2 18275.679} C_VEL
LIN {X 0,Y 383.826,Z 1285.179,A -85,B 0,C 180,E1 18280.761,E2 18280.761} C_VEL
LIN {X 0,Y 385.303,Z 1269.177,A -85,B 0,C 180,E1 18286.283,E2 18286.283} C_VEL
LIN {X 0,Y 388.446,Z 1247.485,A -85,B 0,C 180,E1 18291.462,E2 18291.462} C_VEL
LIN {X 0,Y 396.603,Z 1211.42,A -85,B 0,C 180,E1 18298.308,E2 18298.308} C_VEL
LIN {X 0,Y 402.754,Z 1188.376,A -85,B 0,C 180,E1 18301.614,E2 18301.614} C_VEL
LIN {X 0,Y 402.89,Z 1176.339,A -85,B 0,C 180,E1 18303.427,E2 18303.427} C_VEL
LIN {X 0,Y 403.218,Z 1163.741,A -85,B 0,C 180,E1 18305.151,E2 18305.151} C_VEL
LIN {X 0,Y 414.118,Z 1124.223,A -85,B 0,C 180,E1 18308.645,E2 18308.645} C_VEL
LIN {X 0,Y 423.714,Z 1083.801,A -85,B 0,C 180,E1 18311.233,E2 18311.233} C_VEL
LIN {X 0,Y 423.042,Z 1067.916,A -85,B 0,C 180,E1 18312.803,E2 18312.803} C_VEL
LIN {X 0,Y 418.604,Z 1049.336,A -85,B 0,C 180,E1 18315.566,E2 18315.566} C_VEL
LIN {X 0,Y 413.478,Z 1035.468,A -85,B 0,C 180,E1 18318.753,E2 18318.753} C_VEL
LIN {X 0,Y 410.477,Z 1029.081,A -85,B 0,C 180,E1 18321.155,E2 18321.155} C_VEL
LIN {X 0,Y 407.65,Z 1023.248,A -85,B 0,C 180,E1 18326.136,E2 18326.136} C_VEL
LIN {X 0,Y 409.271,Z 1029.8,A -85,B 0,C 180,E1 18331.93,E2 18331.93} C_VEL
LIN {X 0,Y 413.402,Z 1039.732,A -85,B 0,C 180,E1 18335.616,E2 18335.616} C_VEL
LIN {X 0,Y 418.935,Z 1056.034,A -85,B 0,C 180,E1 18339.214,E2 18339.214} C_VEL
LIN {X 0,Y 421.306,Z 1066.749,A -85,B 0,C 180,E1 18340.809,E2 18340.809} C_VEL
LIN {X 0,Y 412.541,Z 1108.095,A -85,B 0,C 180,E1 18343.239,E2 18343.239} C_VEL
LIN {X 0,Y 405.348,Z 1136.067,A -85,B 0,C 180,E1 18345.817,E2 18345.817} C_VEL
LIN {X 0,Y 397.235,Z 1161.18,A -85,B 0,C 180,E1 18349.3,E2 18349.3} C_VEL
LIN {X 0,Y 390.127,Z 1180.083,A -85,B 0,C 180,E1 18353.325,E2 18353.325} C_VEL
LIN {X 0,Y 384.472,Z 1193.026,A -85,B 0,C 180,E1 18357.758,E2 18357.758} C_VEL
LIN {X 0,Y 380.557,Z 1200.072,A -85,B 0,C 180,E1 18362.298,E2 18362.298} C_VEL
LIN {X 0,Y 378.21,Z 1201.592,A -85,B 0,C 180,E1 18366.919,E2 18366.919} C_VEL
LIN {X 0,Y 377.543,Z 1197.567,A -85,B 0,C 180,E1 18371.592,E2 18371.592} C_VEL
LIN {X 0,Y 378.059,Z 1187.474,A -85,B 0,C 180,E1 18376.309,E2 18376.309} C_VEL
LIN {X 0,Y 379.622,Z 1171.687,A -85,B 0,C 180,E1 18380.679,E2 18380.679} C_VEL
LIN {X 0,Y 381.984,Z 1150.524,A -85,B 0,C 180,E1 18384.572,E2 18384.572} C_VEL
LIN {X 0,Y 384.768,Z 1125.541,A -85,B 0,C 180,E1 18387.716,E2 18387.716} C_VEL
LIN {X 0,Y 387.559,Z 1096.76,A -85,B 0,C 180,E1 18390.158,E2 18390.158} C_VEL
LIN {X 0,Y 389.577,Z 1065.006,A -85,B 0,C 180,E1 18391.793,E2 18391.793} C_VEL
LIN {X 0,Y 390.056,Z 1037.279,A -85,B 0,C 180,E1 18392.806,E2 18392.806} C_VEL
LIN {X 0,Y 373.063,Z 977.53,A -85,B 0,C 180,E1 18396.084,E2 18396.084} C_VEL
LIN {X 0,Y 372.794,Z 977.53,A -85,B 0,C 180,E1 18403.725,E2 18403.725} C_VEL
LIN {X 0,Y 372.766,Z 977.53,A -85,B 0,C 180,E1 18410.582,E2 18410.582} C_VEL
LIN {X 0,Y 373.044,Z 977.53,A -85,B 0,C 180,E1 18418.56,E2 18418.56} C_VEL
LIN {X 0,Y 373.442,Z 977.53,A -85,B 0,C 180,E1 18426.05,E2 18426.05} C_VEL
LIN {X 0,Y 373.822,Z 977.53,A -85,B 0,C 180,E1 18433.505,E2 18433.505} C_VEL
LIN {X 0,Y 374.286,Z 977.53,A -85,B 0,C 180,E1 18440.67,E2 18440.67} C_VEL
LIN {X 0,Y 374.862,Z 977.53,A -85,B 0,C 180,E1 18447.673,E2 18447.673} C_VEL
LIN {X 0,Y 374.887,Z 977.53,A -85,B 0,C 180,E1 18452.306,E2 18452.306} C_VEL
LIN {X 0,Y 374.263,Z 977.53,A -85,B 0,C 180,E1 18459.309,E2 18459.309} C_VEL
LIN {X 0,Y 373.795,Z 977.53,A -85,B 0,C 180,E1 18466.473,E2 18466.473} C_VEL
LIN {X 0,Y 373.402,Z 977.53,A -85,B 0,C 180,E1 18473.929,E2 18473.929} C_VEL
LIN {X 0,Y 373.038,Z 977.53,A -85,B 0,C 180,E1 18481.861,E2 18481.861} C_VEL
LIN {X 0,Y 372.827,Z 977.53,A -85,B 0,C 180,E1 18489.429,E2 18489.429} C_VEL
LIN {X 0,Y 372.921,Z 977.93,A -85,B 0,C 180,E1 18496.294,E2 18496.294} C_VEL
LIN {X 0,Y 395.04,Z 1034.8,A -85,B 0,C 180,E1 18500.082,E2 18500.082} C_VEL
LIN {X 0,Y 407.052,Z 1073.3,A -85,B 0,C 180,E1 18503.016,E2 18503.016} C_VEL
LIN {X 0,Y 401.125,Z 1112.09,A -85,B 0,C 180,E1 18505.582,E2 18505.582} C_VEL
LIN {X 0,Y 394.593,Z 1148.222,A -85,B 0,C 180,E1 18508.921,E2 18508.921} C_VEL
LIN {X 0,Y 388.181,Z 1181.216,A -85,B 0,C 180,E1 18513.093,E2 18513.093} C_VEL
LIN {X 0,Y 382.751,Z 1208.576,A -85,B 0,C 180,E1 18517.802,E2 18517.802} C_VEL
LIN {X 0,Y 378.972,Z 1230.093,A -85,B 0,C 180,E1 18522.835,E2 18522.835} C_VEL
LIN {X 0,Y 376.801,Z 1245.453,A -85,B 0,C 180,E1 18527.796,E2 18527.796} C_VEL
LIN {X 0,Y 375.67,Z 1256.46,A -85,B 0,C 180,E1 18533.034,E2 18533.034} C_VEL
LIN {X 0,Y 375.395,Z 1262.172,A -85,B 0,C 180,E1 18537.67,E2 18537.67} C_VEL
LIN {X 0,Y 375.599,Z 1264.499,A -85,B 0,C 180,E1 18542.295,E2 18542.295} C_VEL
LIN {X 0,Y 376.221,Z 1263.334,A -85,B 0,C 180,E1 18546.922,E2 18546.922} C_VEL
LIN {X 0,Y 378.233,Z 1257.318,A -85,B 0,C 180,E1 18552.711,E2 18552.711} C_VEL
LIN {X 0,Y 382.426,Z 1245.966,A -85,B 0,C 180,E1 18558.461,E2 18558.461} C_VEL
LIN {X 0,Y 389.371,Z 1228.805,A -85,B 0,C 180,E1 18564.112,E2 18564.112} C_VEL
LIN {X 0,Y 399.567,Z 1205.191,A -85,B 0,C 180,E1 18569.516,E2 18569.516} C_VEL
LIN {X 0,Y 412.435,Z 1175.343,A -85,B 0,C 180,E1 18574.37,E2 18574.37} C_VEL
LIN {X 0,Y 427.315,Z 1140.573,A -85,B 0,C 180,E1 18578.465,E2 18578.465} C_VEL
LIN {X 0,Y 442.841,Z 1103.117,A -85,B 0,C 180,E1 18581.612,E2 18581.612} C_VEL
LIN {X 0,Y 448.175,Z 1089.695,A -85,B 0,C 180,E1 18582.522,E2 18582.522} C_VEL
LIN {X 0,Y 449.298,Z 1085.196,A -85,B 0,C 180,E1 18583.715,E2 18583.715} C_VEL
LIN {X 0,Y 449.699,Z 1084.391,A -85,B 0,C 180,E1 18585.013,E2 18585.013} C_VEL
LIN {X 0,Y 449.105,Z 1086.72,A -85,B 0,C 180,E1 18585.629,E2 18585.629} C_VEL
LIN {X 0,Y 445.97,Z 1096.475,A -85,B 0,C 180,E1 18586.683,E2 18586.683} C_VEL
LIN {X 0,Y 429.736,Z 1137.318,A -85,B 0,C 180,E1 18589.312,E2 18589.312} C_VEL
LIN {X 0,Y 412.938,Z 1179.344,A -85,B 0,C 180,E1 18593.244,E2 18593.244} C_VEL
LIN {X 0,Y 399.922,Z 1213.155,A -85,B 0,C 180,E1 18597.656,E2 18597.656} C_VEL
LIN {X 0,Y 389.415,Z 1242.146,A -85,B 0,C 180,E1 18602.774,E2 18602.774} C_VEL
LIN {X 0,Y 382.026,Z 1264.83,A -85,B 0,C 180,E1 18608.269,E2 18608.269} C_VEL
LIN {X 0,Y 377.463,Z 1282.392,A -85,B 0,C 180,E1 18614.374,E2 18614.374} C_VEL
LIN {X 0,Y 375.857,Z 1292.178,A -85,B 0,C 180,E1 18619.559,E2 18619.559} C_VEL
LIN {X 0,Y 375.443,Z 1297.865,A -85,B 0,C 180,E1 18625.381,E2 18625.381} C_VEL
LIN {X 0,Y 375.699,Z 1298.33,A -85,B 0,C 180,E1 18630.011,E2 18630.011} C_VEL
LIN {X 0,Y 375.589,Z 1295.036,A -85,B 0,C 180,E1 18634.639,E2 18634.639} C_VEL
LIN {X 0,Y 375.842,Z 1286.643,A -85,B 0,C 180,E1 18639.877,E2 18639.877} C_VEL
LIN {X 0,Y 376.996,Z 1273.127,A -85,B 0,C 180,E1 18645.062,E2 18645.062} C_VEL
LIN {X 0,Y 379.677,Z 1253.24,A -85,B 0,C 180,E1 18650.34,E2 18650.34} C_VEL
LIN {X 0,Y 387.654,Z 1218.395,A -85,B 0,C 180,E1 18657.668,E2 18657.668} C_VEL
LIN {X 0,Y 396.388,Z 1187.568,A -85,B 0,C 180,E1 18662.368,E2 18662.368} C_VEL
LIN {X 0,Y 403.218,Z 1163.741,A -85,B 0,C 180,E1 18665.151,E2 18665.151} C_VEL
LIN {X 0,Y 403.88,Z 1150.806,A -85,B 0,C 180,E1 18666.843,E2 18666.843} C_VEL
LIN {X 0,Y 404.409,Z 1139.231,A -85,B 0,C 180,E1 18668.267,E2 18668.267} C_VEL
LIN {X 0,Y 404.882,Z 1137.407,A -85,B 0,C 180,E1 18668.426,E2 18668.426} C_VEL
LIN {X 0,Y 416.82,Z 1094.375,A -85,B 0,C 180,E1 18671.428,E2 18671.428} C_VEL
LIN {X 0,Y 418.413,Z 1085.704,A -85,B 0,C 180,E1 18672.007,E2 18672.007} C_VEL
LIN {X 0,Y 417.934,Z 1071.113,A -85,B 0,C 180,E1 18673.554,E2 18673.554} C_VEL
LIN {X 0,Y 414.129,Z 1053.82,A -85,B 0,C 180,E1 18676.316,E2 18676.316} C_VEL
LIN {X 0,Y 410.006,Z 1041.688,A -85,B 0,C 180,E1 18679.292,E2 18679.292} C_VEL
LIN {X 0,Y 407.729,Z 1036.443,A -85,B 0,C 180,E1 18681.316,E2 18681.316} C_VEL
LIN {X 0,Y 405.078,Z 1031.013,A -85,B 0,C 180,E1 18685.891,E2 18685.891} C_VEL
LIN {X 0,Y 405.807,Z 1035.551,A -85,B 0,C 180,E1 18690.982,E2 18690.982} C_VEL
LIN {X 0,Y 409.519,Z 1045.603,A -85,B 0,C 180,E1 18695.066,E2 18695.066} C_VEL
LIN {X 0,Y 414.242,Z 1060.594,A -85,B 0,C 180,E1 18698.562,E2 18698.562} C_VEL
LIN {X 0,Y 416,Z 1070.629,A -85,B 0,C 180,E1 18700.09,E2 18700.09} C_VEL
LIN {X 0,Y 406.876,Z 1110.661,A -85,B 0,C 180,E1 18702.545,E2 18702.545} C_VEL
LIN {X 0,Y 399.212,Z 1138.159,A -85,B 0,C 180,E1 18705.173,E2 18705.173} C_VEL
LIN {X 0,Y 391.018,Z 1161.971,A -85,B 0,C 180,E1 18708.562,E2 18708.562} C_VEL
LIN {X 0,Y 383.836,Z 1179.865,A -85,B 0,C 180,E1 18712.361,E2 18712.361} C_VEL
LIN {X 0,Y 378.051,Z 1192.676,A -85,B 0,C 180,E1 18716.57,E2 18716.57} C_VEL
LIN {X 0,Y 373.531,Z 1200.454,A -85,B 0,C 180,E1 18721.179,E2 18721.179} C_VEL
LIN {X 0,Y 371.326,Z 1202.725,A -85,B 0,C 180,E1 18724.698,E2 18724.698} C_VEL
LIN {X 0,Y 369.831,Z 1200.957,A -85,B 0,C 180,E1 18729.448,E2 18729.448} C_VEL
LIN {X 0,Y 369.864,Z 1193.419,A -85,B 0,C 180,E1 18734.245,E2 18734.245} C_VEL
LIN {X 0,Y 370.89,Z 1180.375,A -85,B 0,C 180,E1 18738.783,E2 18738.783} C_VEL
LIN {X 0,Y 372.95,Z 1161.379,A -85,B 0,C 180,E1 18743.035,E2 18743.035} C_VEL
LIN {X 0,Y 375.719,Z 1138.317,A -85,B 0,C 180,E1 18746.539,E2 18746.539} C_VEL
LIN {X 0,Y 378.567,Z 1111.219,A -85,B 0,C 180,E1 18749.377,E2 18749.377} C_VEL
LIN {X 0,Y 381.121,Z 1080.853,A -85,B 0,C 180,E1 18751.428,E2 18751.428} C_VEL
LIN {X 0,Y 382.67,Z 1039.271,A -85,B 0,C 180,E1 18753.105,E2 18753.105} C_VEL
LIN {X 0,Y 365.108,Z 977.53,A -85,B 0,C 180,E1 18756.557,E2 18756.557} C_VEL
LIN {X 0,Y 364.857,Z 977.53,A -85,B 0,C 180,E1 18761.66,E2 18761.66} C_VEL
LIN {X 0,Y 364.804,Z 977.53,A -85,B 0,C 180,E1 18768.406,E2 18768.406} C_VEL
LIN {X 0,Y 364.907,Z 977.53,A -85,B 0,C 180,E1 18774.441,E2 18774.441} C_VEL
LIN {X 0,Y 365.213,Z 977.53,A -85,B 0,C 180,E1 18780.631,E2 18780.631} C_VEL
LIN {X 0,Y 365.577,Z 977.53,A -85,B 0,C 180,E1 18788.085,E2 18788.085} C_VEL
LIN {X 0,Y 366.021,Z 977.53,A -85,B 0,C 180,E1 18795.606,E2 18795.606} C_VEL
LIN {X 0,Y 366.589,Z 977.53,A -85,B 0,C 180,E1 18802.866,E2 18802.866} C_VEL
LIN {X 0,Y 367.17,Z 977.53,A -85,B 0,C 180,E1 18809.989,E2 18809.989} C_VEL
LIN {X 0,Y 366.549,Z 977.53,A -85,B 0,C 180,E1 18817.113,E2 18817.113} C_VEL
LIN {X 0,Y 366.014,Z 977.53,A -85,B 0,C 180,E1 18824.371,E2 18824.371} C_VEL
LIN {X 0,Y 365.564,Z 977.53,A -85,B 0,C 180,E1 18831.892,E2 18831.892} C_VEL
LIN {X 0,Y 365.157,Z 977.53,A -85,B 0,C 180,E1 18839.852,E2 18839.852} C_VEL
LIN {X 0,Y 364.955,Z 977.53,A -85,B 0,C 180,E1 18845.526,E2 18845.526} C_VEL
LIN {X 0,Y 364.846,Z 977.53,A -85,B 0,C 180,E1 18851.629,E2 18851.629} C_VEL
LIN {X 0,Y 364.959,Z 977.53,A -85,B 0,C 180,E1 18855.551,E2 18855.551} C_VEL
LIN {X 0,Y 387.487,Z 1035.851,A -85,B 0,C 180,E1 18859.565,E2 18859.565} C_VEL
LIN {X 0,Y 399.559,Z 1073.863,A -85,B 0,C 180,E1 18862.55,E2 18862.55} C_VEL
LIN {X 0,Y 393.598,Z 1113.677,A -85,B 0,C 180,E1 18865.266,E2 18865.266} C_VEL
LIN {X 0,Y 386.865,Z 1150.037,A -85,B 0,C 180,E1 18868.722,E2 18868.722} C_VEL
LIN {X 0,Y 380.223,Z 1182.999,A -85,B 0,C 180,E1 18873.028,E2 18873.028} C_VEL
LIN {X 0,Y 374.875,Z 1209.495,A -85,B 0,C 180,E1 18877.717,E2 18877.717} C_VEL
LIN {X 0,Y 371.094,Z 1230.589,A -85,B 0,C 180,E1 18882.765,E2 18882.765} C_VEL
LIN {X 0,Y 368.815,Z 1246.676,A -85,B 0,C 180,E1 18888.13,E2 18888.13} C_VEL
LIN {X 0,Y 367.797,Z 1256.488,A -85,B 0,C 180,E1 18892.884,E2 18892.884} C_VEL
LIN {X 0,Y 367.498,Z 1262.385,A -85,B 0,C 180,E1 18897.62,E2 18897.62} C_VEL
LIN {X 0,Y 367.707,Z 1264.889,A -85,B 0,C 180,E1 18902.345,E2 18902.345} C_VEL
LIN {X 0,Y 368.396,Z 1263.969,A -85,B 0,C 180,E1 18907.07,E2 18907.07} C_VEL
LIN {X 0,Y 370.548,Z 1258.24,A -85,B 0,C 180,E1 18912.979,E2 18912.979} C_VEL
LIN {X 0,Y 375.019,Z 1247.239,A -85,B 0,C 180,E1 18918.839,E2 18918.839} C_VEL
LIN {X 0,Y 382.413,Z 1230.408,A -85,B 0,C 180,E1 18924.622,E2 18924.622} C_VEL
LIN {X 0,Y 393.678,Z 1206.31,A -85,B 0,C 180,E1 18930.321,E2 18930.321} C_VEL
LIN {X 0,Y 408.218,Z 1175.277,A -85,B 0,C 180,E1 18935.456,E2 18935.456} C_VEL
LIN {X 0,Y 424.597,Z 1140.194,A -85,B 0,C 180,E1 18939.603,E2 18939.603} C_VEL
LIN {X 0,Y 441.917,Z 1102.167,A -85,B 0,C 180,E1 18942.767,E2 18942.767} C_VEL
LIN {X 0,Y 445.375,Z 1094.158,A -85,B 0,C 180,E1 18943.338,E2 18943.338} C_VEL
LIN {X 0,Y 446.237,Z 1091.872,A -85,B 0,C 180,E1 18944.526,E2 18944.526} C_VEL
LIN {X 0,Y 446,Z 1092.776,A -85,B 0,C 180,E1 18945.047,E2 18945.047} C_VEL
LIN {X 0,Y 443.222,Z 1099.884,A -85,B 0,C 180,E1 18945.815,E2 18945.815} C_VEL
LIN {X 0,Y 425.128,Z 1141.314,A -85,B 0,C 180,E1 18948.589,E2 18948.589} C_VEL
LIN {X 0,Y 407.044,Z 1182.539,A -85,B 0,C 180,E1 18952.622,E2 18952.622} C_VEL
LIN {X 0,Y 392.129,Z 1218.28,A -85,B 0,C 180,E1 18957.578,E2 18957.578} C_VEL
LIN {X 0,Y 381.439,Z 1245.807,A -85,B 0,C 180,E1 18962.829,E2 18962.829} C_VEL
LIN {X 0,Y 374.384,Z 1265.947,A -85,B 0,C 180,E1 18968.026,E2 18968.026} C_VEL
LIN {X 0,Y 369.643,Z 1282.943,A -85,B 0,C 180,E1 18974.254,E2 18974.254} C_VEL
LIN {X 0,Y 367.885,Z 1293.537,A -85,B 0,C 180,E1 18980.528,E2 18980.528} C_VEL
LIN {X 0,Y 367.538,Z 1297.54,A -85,B 0,C 180,E1 18985.281,E2 18985.281} C_VEL
LIN {X 0,Y 367.813,Z 1297.808,A -85,B 0,C 180,E1 18990.011,E2 18990.011} C_VEL
LIN {X 0,Y 367.708,Z 1294.379,A -85,B 0,C 180,E1 18994.738,E2 18994.738} C_VEL
LIN {X 0,Y 367.986,Z 1285.743,A -85,B 0,C 180,E1 19000.09,E2 19000.09} C_VEL
LIN {X 0,Y 369.183,Z 1271.939,A -85,B 0,C 180,E1 19005.389,E2 19005.389} C_VEL
LIN {X 0,Y 372.093,Z 1251.461,A -85,B 0,C 180,E1 19010.839,E2 19010.839} C_VEL
LIN {X 0,Y 378.732,Z 1224.484,A -85,B 0,C 180,E1 19017.083,E2 19017.083} C_VEL
LIN {X 0,Y 387.862,Z 1194.077,A -85,B 0,C 180,E1 19022.172,E2 19022.172} C_VEL
LIN {X 0,Y 397.944,Z 1161.169,A -85,B 0,C 180,E1 19026.184,E2 19026.184} C_VEL
LIN {X 0,Y 404.882,Z 1137.407,A -85,B 0,C 180,E1 19028.426,E2 19028.426} C_VEL
LIN {X 0,Y 406.35,Z 1123.589,A -85,B 0,C 180,E1 19029.94,E2 19029.94} C_VEL
LIN {X 0,Y 407.863,Z 1109.439,A -85,B 0,C 180,E1 19031.372,E2 19031.372} C_VEL
LIN {X 0,Y 413.243,Z 1088.327,A -85,B 0,C 180,E1 19032.746,E2 19032.746} C_VEL
LIN {X 0,Y 413.113,Z 1075.37,A -85,B 0,C 180,E1 19034.193,E2 19034.193} C_VEL
LIN {X 0,Y 410.08,Z 1059.337,A -85,B 0,C 180,E1 19036.879,E2 19036.879} C_VEL
LIN {X 0,Y 406.927,Z 1048.894,A -85,B 0,C 180,E1 19039.481,E2 19039.481} C_VEL
LIN {X 0,Y 404.364,Z 1043.218,A -85,B 0,C 180,E1 19041.915,E2 19041.915} C_VEL
LIN {X 0,Y 402.4,Z 1038.528,A -85,B 0,C 180,E1 19045.955,E2 19045.955} C_VEL
LIN {X 0,Y 402.81,Z 1042.695,A -85,B 0,C 180,E1 19050.745,E2 19050.745} C_VEL
LIN {X 0,Y 405.521,Z 1051.088,A -85,B 0,C 180,E1 19054.353,E2 19054.353} C_VEL
LIN {X 0,Y 409.413,Z 1064.391,A -85,B 0,C 180,E1 19057.734,E2 19057.734} C_VEL
LIN {X 0,Y 411.141,Z 1073.373,A -85,B 0,C 180,E1 19059.285,E2 19059.285} C_VEL
LIN {X 0,Y 401.177,Z 1113.778,A -85,B 0,C 180,E1 19061.862,E2 19061.862} C_VEL
LIN {X 0,Y 392.621,Z 1141.996,A -85,B 0,C 180,E1 19064.71,E2 19064.71} C_VEL
LIN {X 0,Y 384.292,Z 1164.471,A -85,B 0,C 180,E1 19068.071,E2 19068.071} C_VEL
LIN {X 0,Y 376.757,Z 1181.84,A -85,B 0,C 180,E1 19071.925,E2 19071.925} C_VEL
LIN {X 0,Y 370.318,Z 1194.859,A -85,B 0,C 180,E1 19076.498,E2 19076.498} C_VEL
LIN {X 0,Y 365.693,Z 1202.07,A -85,B 0,C 180,E1 19081.204,E2 19081.204} C_VEL
LIN {X 0,Y 363.435,Z 1203.89,A -85,B 0,C 180,E1 19084.8,E2 19084.8} C_VEL
LIN {X 0,Y 361.941,Z 1201.546,A -85,B 0,C 180,E1 19089.656,E2 19089.656} C_VEL
LIN {X 0,Y 362.035,Z 1193.49,A -85,B 0,C 180,E1 19094.56,E2 19094.56} C_VEL
LIN {X 0,Y 363.138,Z 1179.772,A -85,B 0,C 180,E1 19099.2,E2 19099.2} C_VEL
LIN {X 0,Y 365.305,Z 1160.453,A -85,B 0,C 180,E1 19103.465,E2 19103.465} C_VEL
LIN {X 0,Y 368.283,Z 1136.273,A -85,B 0,C 180,E1 19107.099,E2 19107.099} C_VEL
LIN {X 0,Y 371.251,Z 1108.582,A -85,B 0,C 180,E1 19109.915,E2 19109.915} C_VEL
LIN {X 0,Y 373.749,Z 1077.834,A -85,B 0,C 180,E1 19111.923,E2 19111.923} C_VEL
LIN {X 0,Y 374.994,Z 1040.284,A -85,B 0,C 180,E1 19113.452,E2 19113.452} C_VEL
LIN {X 0,Y 357.161,Z 977.53,A -85,B 0,C 180,E1 19117.027,E2 19117.027} C_VEL
LIN {X 0,Y 356.792,Z 977.53,A -85,B 0,C 180,E1 19123.766,E2 19123.766} C_VEL
LIN {X 0,Y 356.805,Z 977.53,A -85,B 0,C 180,E1 19130.416,E2 19130.416} C_VEL
LIN {X 0,Y 357.031,Z 977.53,A -85,B 0,C 180,E1 19136.501,E2 19136.501} C_VEL
LIN {X 0,Y 357.375,Z 977.53,A -85,B 0,C 180,E1 19142.948,E2 19142.948} C_VEL
LIN {X 0,Y 357.749,Z 977.53,A -85,B 0,C 180,E1 19150.182,E2 19150.182} C_VEL
LIN {X 0,Y 358.234,Z 977.53,A -85,B 0,C 180,E1 19157.779,E2 19157.779} C_VEL
LIN {X 0,Y 358.878,Z 977.53,A -85,B 0,C 180,E1 19165.145,E2 19165.145} C_VEL
LIN {X 0,Y 359.28,Z 977.53,A -85,B 0,C 180,E1 19169.989,E2 19169.989} C_VEL
LIN {X 0,Y 358.611,Z 977.53,A -85,B 0,C 180,E1 19177.271,E2 19177.271} C_VEL
LIN {X 0,Y 358.06,Z 977.53,A -85,B 0,C 180,E1 19184.697,E2 19184.697} C_VEL
LIN {X 0,Y 357.615,Z 977.53,A -85,B 0,C 180,E1 19192.405,E2 19192.405} C_VEL
LIN {X 0,Y 357.303,Z 977.53,A -85,B 0,C 180,E1 19197.794,E2 19197.794} C_VEL
LIN {X 0,Y 357.066,Z 977.53,A -85,B 0,C 180,E1 19203.468,E2 19203.468} C_VEL
LIN {X 0,Y 356.841,Z 977.53,A -85,B 0,C 180,E1 19210.133,E2 19210.133} C_VEL
LIN {X 0,Y 356.975,Z 977.607,A -85,B 0,C 180,E1 19214.827,E2 19214.827} C_VEL
LIN {X 0,Y 379.377,Z 1035.393,A -85,B 0,C 180,E1 19218.912,E2 19218.912} C_VEL
LIN {X 0,Y 392.057,Z 1075.239,A -85,B 0,C 180,E1 19222.129,E2 19222.129} C_VEL
LIN {X 0,Y 386.241,Z 1114.239,A -85,B 0,C 180,E1 19224.861,E2 19224.861} C_VEL
LIN {X 0,Y 379.092,Z 1151.776,A -85,B 0,C 180,E1 19228.51,E2 19228.51} C_VEL
LIN {X 0,Y 372.557,Z 1183.442,A -85,B 0,C 180,E1 19232.755,E2 19232.755} C_VEL
LIN {X 0,Y 367.072,Z 1209.949,A -85,B 0,C 180,E1 19237.537,E2 19237.537} C_VEL
LIN {X 0,Y 363.245,Z 1231.057,A -85,B 0,C 180,E1 19242.694,E2 19242.694} C_VEL
LIN {X 0,Y 360.855,Z 1247.881,A -85,B 0,C 180,E1 19248.479,E2 19248.479} C_VEL
LIN {X 0,Y 359.787,Z 1258.285,A -85,B 0,C 180,E1 19253.94,E2 19253.94} C_VEL
LIN {X 0,Y 359.727,Z 1264.339,A -85,B 0,C 180,E1 19259.983,E2 19259.983} C_VEL
LIN {X 0,Y 360.046,Z 1265.386,A -85,B 0,C 180,E1 19264.81,E2 19264.81} C_VEL
LIN {X 0,Y 361.539,Z 1262.435,A -85,B 0,C 180,E1 19270.307,E2 19270.307} C_VEL
LIN {X 0,Y 365.268,Z 1253.472,A -85,B 0,C 180,E1 19276.861,E2 19276.861} C_VEL
LIN {X 0,Y 372.663,Z 1237.857,A -85,B 0,C 180,E1 19283.335,E2 19283.335} C_VEL
LIN {X 0,Y 382.883,Z 1217.426,A -85,B 0,C 180,E1 19288.993,E2 19288.993} C_VEL
LIN {X 0,Y 396.682,Z 1190.572,A -85,B 0,C 180,E1 19294.253,E2 19294.253} C_VEL
LIN {X 0,Y 413.409,Z 1157.683,A -85,B 0,C 180,E1 19298.854,E2 19298.854} C_VEL
LIN {X 0,Y 431.88,Z 1121.344,A -85,B 0,C 180,E1 19302.459,E2 19302.459} C_VEL
LIN {X 0,Y 442.612,Z 1099.503,A -85,B 0,C 180,E1 19304.11,E2 19304.11} C_VEL
LIN {X 0,Y 441.846,Z 1101.296,A -85,B 0,C 180,E1 19304.754,E2 19304.754} C_VEL
LIN {X 0,Y 419.993,Z 1146.747,A -85,B 0,C 180,E1 19307.968,E2 19307.968} C_VEL
LIN {X 0,Y 400.825,Z 1186.821,A -85,B 0,C 180,E1 19312.111,E2 19312.111} C_VEL
LIN {X 0,Y 384.961,Z 1221.776,A -85,B 0,C 180,E1 19317.246,E2 19317.246} C_VEL
LIN {X 0,Y 373.508,Z 1249.33,A -85,B 0,C 180,E1 19322.857,E2 19322.857} C_VEL
LIN {X 0,Y 365.478,Z 1271.087,A -85,B 0,C 180,E1 19329.091,E2 19329.091} C_VEL
LIN {X 0,Y 361.163,Z 1286.055,A -85,B 0,C 180,E1 19335.432,E2 19335.432} C_VEL
LIN {X 0,Y 359.871,Z 1294.478,A -85,B 0,C 180,E1 19341.369,E2 19341.369} C_VEL
LIN {X 0,Y 359.646,Z 1297.159,A -85,B 0,C 180,E1 19345.178,E2 19345.178} C_VEL
LIN {X 0,Y 359.947,Z 1297.28,A -85,B 0,C 180,E1 19350.011,E2 19350.011} C_VEL
LIN {X 0,Y 359.849,Z 1293.709,A -85,B 0,C 180,E1 19354.842,E2 19354.842} C_VEL
LIN {X 0,Y 360.127,Z 1284.82,A -85,B 0,C 180,E1 19360.313,E2 19360.313} C_VEL
LIN {X 0,Y 361.526,Z 1269.828,A -85,B 0,C 180,E1 19366.023,E2 19366.023} C_VEL
LIN {X 0,Y 369.501,Z 1231.811,A -85,B 0,C 180,E1 19376.077,E2 19376.077} C_VEL
LIN {X 0,Y 378.195,Z 1203.74,A -85,B 0,C 180,E1 19381.402,E2 19381.402} C_VEL
LIN {X 0,Y 388.587,Z 1171.781,A -85,B 0,C 180,E1 19385.81,E2 19385.81} C_VEL
LIN {X 0,Y 400.612,Z 1133.718,A -85,B 0,C 180,E1 19389.574,E2 19389.574} C_VEL
LIN {X 0,Y 407.863,Z 1109.439,A -85,B 0,C 180,E1 19391.372,E2 19391.372} C_VEL
LIN {X 0,Y 408.529,Z 1100.114,A -85,B 0,C 180,E1 19392.361,E2 19392.361} C_VEL
LIN {X 0,Y 408.182,Z 1091.181,A -85,B 0,C 180,E1 19393.493,E2 19393.493} C_VEL
LIN {X 0,Y 408.265,Z 1078.661,A -85,B 0,C 180,E1 19394.983,E2 19394.983} C_VEL
LIN {X 0,Y 405.639,Z 1063.243,A -85,B 0,C 180,E1 19397.775,E2 19397.775} C_VEL
LIN {X 0,Y 403.002,Z 1054.391,A -85,B 0,C 180,E1 19400.294,E2 19400.294} C_VEL
LIN {X 0,Y 400.741,Z 1049.569,A -85,B 0,C 180,E1 19402.797,E2 19402.797} C_VEL
LIN {X 0,Y 399.658,Z 1046.543,A -85,B 0,C 180,E1 19405.363,E2 19405.363} C_VEL
LIN {X 0,Y 399.07,Z 1047.285,A -85,B 0,C 180,E1 19407.91,E2 19407.91} C_VEL
LIN {X 0,Y 400.347,Z 1052.364,A -85,B 0,C 180,E1 19411.84,E2 19411.84} C_VEL
LIN {X 0,Y 403.438,Z 1063.104,A -85,B 0,C 180,E1 19415.617,E2 19415.617} C_VEL
LIN {X 0,Y 406.362,Z 1076.666,A -85,B 0,C 180,E1 19418.479,E2 19418.479} C_VEL
LIN {X 0,Y 396.031,Z 1115.435,A -85,B 0,C 180,E1 19421.04,E2 19421.04} C_VEL
LIN {X 0,Y 387.176,Z 1142.815,A -85,B 0,C 180,E1 19423.845,E2 19423.845} C_VEL
LIN {X 0,Y 378.217,Z 1165.5,A -85,B 0,C 180,E1 19427.289,E2 19427.289} C_VEL
LIN {X 0,Y 370.224,Z 1182.786,A -85,B 0,C 180,E1 19431.189,E2 19431.189} C_VEL
LIN {X 0,Y 363.334,Z 1195.839,A -85,B 0,C 180,E1 19435.832,E2 19435.832} C_VEL
LIN {X 0,Y 358.866,Z 1202.476,A -85,B 0,C 180,E1 19440.017,E2 19440.017} C_VEL
LIN {X 0,Y 355.534,Z 1204.986,A -85,B 0,C 180,E1 19444.907,E2 19444.907} C_VEL
LIN {X 0,Y 354.064,Z 1201.844,A -85,B 0,C 180,E1 19450.097,E2 19450.097} C_VEL
LIN {X 0,Y 354.185,Z 1193.44,A -85,B 0,C 180,E1 19454.89,E2 19454.89} C_VEL
LIN {X 0,Y 355.416,Z 1179.137,A -85,B 0,C 180,E1 19459.634,E2 19459.634} C_VEL
LIN {X 0,Y 357.699,Z 1159.535,A -85,B 0,C 180,E1 19463.892,E2 19463.892} C_VEL
LIN {X 0,Y 360.727,Z 1135.084,A -85,B 0,C 180,E1 19467.536,E2 19467.536} C_VEL
LIN {X 0,Y 363.862,Z 1106.688,A -85,B 0,C 180,E1 19470.41,E2 19470.41} C_VEL
LIN {X 0,Y 366.396,Z 1074.639,A -85,B 0,C 180,E1 19472.435,E2 19472.435} C_VEL
LIN {X 0,Y 367.641,Z 1042.333,A -85,B 0,C 180,E1 19473.752,E2 19473.752} C_VEL
LIN {X 0,Y 349.213,Z 977.53,A -85,B 0,C 180,E1 19477.619,E2 19477.619} C_VEL
LIN {X 0,Y 348.848,Z 977.53,A -85,B 0,C 180,E1 19485.958,E2 19485.958} C_VEL
LIN {X 0,Y 348.874,Z 977.53,A -85,B 0,C 180,E1 19492.536,E2 19492.536} C_VEL
LIN {X 0,Y 349.189,Z 977.53,A -85,B 0,C 180,E1 19500.237,E2 19500.237} C_VEL
LIN {X 0,Y 349.631,Z 977.53,A -85,B 0,C 180,E1 19507.03,E2 19507.03} C_VEL
LIN {X 0,Y 350.11,Z 977.53,A -85,B 0,C 180,E1 19514.937,E2 19514.937} C_VEL
LIN {X 0,Y 350.749,Z 977.53,A -85,B 0,C 180,E1 19522.542,E2 19522.542} C_VEL
LIN {X 0,Y 351.375,Z 977.53,A -85,B 0,C 180,E1 19529.989,E2 19529.989} C_VEL
LIN {X 0,Y 350.694,Z 977.53,A -85,B 0,C 180,E1 19537.436,E2 19537.436} C_VEL
LIN {X 0,Y 350.095,Z 977.53,A -85,B 0,C 180,E1 19545.04,E2 19545.04} C_VEL
LIN {X 0,Y 349.607,Z 977.53,A -85,B 0,C 180,E1 19552.947,E2 19552.947} C_VEL
LIN {X 0,Y 349.195,Z 977.53,A -85,B 0,C 180,E1 19559.765,E2 19559.765} C_VEL
LIN {X 0,Y 348.942,Z 977.53,A -85,B 0,C 180,E1 19567.426,E2 19567.426} C_VEL
LIN {X 0,Y 348.992,Z 977.53,A -85,B 0,C 180,E1 19574.051,E2 19574.051} C_VEL
LIN {X 0,Y 371.874,Z 1036.476,A -85,B 0,C 180,E1 19578.373,E2 19578.373} C_VEL
LIN {X 0,Y 384.245,Z 1075.311,A -85,B 0,C 180,E1 19581.589,E2 19581.589} C_VEL
LIN {X 0,Y 384.067,Z 1083.92,A -85,B 0,C 180,E1 19582.182,E2 19582.182} C_VEL
LIN {X 0,Y 377.12,Z 1124.11,A -85,B 0,C 180,E1 19585.263,E2 19585.263} C_VEL
LIN {X 0,Y 370.166,Z 1159.03,A -85,B 0,C 180,E1 19588.992,E2 19588.992} C_VEL
LIN {X 0,Y 363.616,Z 1190.128,A -85,B 0,C 180,E1 19593.501,E2 19593.501} C_VEL
LIN {X 0,Y 358.022,Z 1217.076,A -85,B 0,C 180,E1 19598.856,E2 19598.856} C_VEL
LIN {X 0,Y 354.446,Z 1237.154,A -85,B 0,C 180,E1 19604.366,E2 19604.366} C_VEL
LIN {X 0,Y 352.535,Z 1251.719,A -85,B 0,C 180,E1 19610.083,E2 19610.083} C_VEL
LIN {X 0,Y 351.758,Z 1261.489,A -85,B 0,C 180,E1 19616.278,E2 19616.278} C_VEL
LIN {X 0,Y 351.923,Z 1265.65,A -85,B 0,C 180,E1 19622.45,E2 19622.45} C_VEL
LIN {X 0,Y 352.754,Z 1265.261,A -85,B 0,C 180,E1 19627.385,E2 19627.385} C_VEL
LIN {X 0,Y 355.191,Z 1260.141,A -85,B 0,C 180,E1 19633.55,E2 19633.55} C_VEL
LIN {X 0,Y 360.925,Z 1248.56,A -85,B 0,C 180,E1 19640.244,E2 19640.244} C_VEL
LIN {X 0,Y 369.455,Z 1232.374,A -85,B 0,C 180,E1 19646.138,E2 19646.138} C_VEL
LIN {X 0,Y 382.27,Z 1209.017,A -85,B 0,C 180,E1 19651.993,E2 19651.993} C_VEL
LIN {X 0,Y 399.403,Z 1178.283,A -85,B 0,C 180,E1 19657.349,E2 19657.349} C_VEL
LIN {X 0,Y 418.234,Z 1144.796,A -85,B 0,C 180,E1 19661.474,E2 19661.474} C_VEL
LIN {X 0,Y 435.784,Z 1112.995,A -85,B 0,C 180,E1 19664.376,E2 19664.376} C_VEL
LIN {X 0,Y 414.923,Z 1152.312,A -85,B 0,C 180,E1 19667.335,E2 19667.335} C_VEL
LIN {X 0,Y 395.086,Z 1190.152,A -85,B 0,C 180,E1 19671.461,E2 19671.461} C_VEL
LIN {X 0,Y 378.562,Z 1223.748,A -85,B 0,C 180,E1 19676.621,E2 19676.621} C_VEL
LIN {X 0,Y 366.511,Z 1250.305,A -85,B 0,C 180,E1 19682.295,E2 19682.295} C_VEL
LIN {X 0,Y 358.18,Z 1271.085,A -85,B 0,C 180,E1 19688.48,E2 19688.48} C_VEL
LIN {X 0,Y 353.424,Z 1286.107,A -85,B 0,C 180,E1 19695.105,E2 19695.105} C_VEL
LIN {X 0,Y 352.126,Z 1293.23,A -85,B 0,C 180,E1 19700.1,E2 19700.1} C_VEL
LIN {X 0,Y 351.744,Z 1296.771,A -85,B 0,C 180,E1 19705.069,E2 19705.069} C_VEL
LIN {X 0,Y 352.061,Z 1296.744,A -85,B 0,C 180,E1 19710.011,E2 19710.011} C_VEL
LIN {X 0,Y 351.969,Z 1292.969,A -85,B 0,C 180,E1 19714.951,E2 19714.951} C_VEL
LIN {X 0,Y 352.292,Z 1283.879,A -85,B 0,C 180,E1 19720.544,E2 19720.544} C_VEL
LIN {X 0,Y 353.838,Z 1267.92,A -85,B 0,C 180,E1 19726.577,E2 19726.577} C_VEL
LIN {X 0,Y 361.743,Z 1233.523,A -85,B 0,C 180,E1 19736.222,E2 19736.222} C_VEL
LIN {X 0,Y 370.296,Z 1207.37,A -85,B 0,C 180,E1 19741.505,E2 19741.505} C_VEL
LIN {X 0,Y 381.513,Z 1175.174,A -85,B 0,C 180,E1 19746.226,E2 19746.226} C_VEL
LIN {X 0,Y 394.275,Z 1137.328,A -85,B 0,C 180,E1 19750.157,E2 19750.157} C_VEL
LIN {X 0,Y 407.268,Z 1095.313,A -85,B 0,C 180,E1 19753.184,E2 19753.184} C_VEL
LIN {X 0,Y 408.182,Z 1091.181,A -85,B 0,C 180,E1 19753.493,E2 19753.493} C_VEL
LIN {X 0,Y 407.443,Z 1083.72,A -85,B 0,C 180,E1 19754.6,E2 19754.6} C_VEL
LIN {X 0,Y 402.217,Z 1072.012,A -85,B 0,C 180,E1 19757.629,E2 19757.629} C_VEL
LIN {X 0,Y 399.569,Z 1060.988,A -85,B 0,C 180,E1 19760.686,E2 19760.686} C_VEL
LIN {X 0,Y 397.103,Z 1055.534,A -85,B 0,C 180,E1 19763.983,E2 19763.983} C_VEL
LIN {X 0,Y 396.792,Z 1054.298,A -85,B 0,C 180,E1 19765.077,E2 19765.077} C_VEL
LIN {X 0,Y 396.147,Z 1054.466,A -85,B 0,C 180,E1 19767.645,E2 19767.645} C_VEL
LIN {X 0,Y 396.973,Z 1058.941,A -85,B 0,C 180,E1 19771.413,E2 19771.413} C_VEL
LIN {X 0,Y 399.299,Z 1068.257,A -85,B 0,C 180,E1 19774.91,E2 19774.91} C_VEL
LIN {X 0,Y 401.483,Z 1080.894,A -85,B 0,C 180,E1 19777.704,E2 19777.704} C_VEL
LIN {X 0,Y 390.548,Z 1118.821,A -85,B 0,C 180,E1 19780.321,E2 19780.321} C_VEL
LIN {X 0,Y 380.857,Z 1146.299,A -85,B 0,C 180,E1 19783.287,E2 19783.287} C_VEL
LIN {X 0,Y 370.918,Z 1169.493,A -85,B 0,C 180,E1 19787.034,E2 19787.034} C_VEL
LIN {X 0,Y 362.737,Z 1185.86,A -85,B 0,C 180,E1 19791.006,E2 19791.006} C_VEL
LIN {X 0,Y 355.628,Z 1198.074,A -85,B 0,C 180,E1 19795.742,E2 19795.742} C_VEL
LIN {X 0,Y 351.029,Z 1204.104,A -85,B 0,C 180,E1 19800.018,E2 19800.018} C_VEL
LIN {X 0,Y 347.654,Z 1206.075,A -85,B 0,C 180,E1 19805.018,E2 19805.018} C_VEL
LIN {X 0,Y 346.205,Z 1202.582,A -85,B 0,C 180,E1 19810.1,E2 19810.1} C_VEL
LIN {X 0,Y 346.365,Z 1193.35,A -85,B 0,C 180,E1 19815.234,E2 19815.234} C_VEL
LIN {X 0,Y 347.73,Z 1178.369,A -85,B 0,C 180,E1 19820.086,E2 19820.086} C_VEL
LIN {X 0,Y 350.084,Z 1158.819,A -85,B 0,C 180,E1 19824.297,E2 19824.297} C_VEL
LIN {X 0,Y 353.158,Z 1133.745,A -85,B 0,C 180,E1 19828.004,E2 19828.004} C_VEL
LIN {X 0,Y 356.466,Z 1104.793,A -85,B 0,C 180,E1 19830.886,E2 19830.886} C_VEL
LIN {X 0,Y 358.897,Z 1073.315,A -85,B 0,C 180,E1 19832.864,E2 19832.864} C_VEL
LIN {X 0,Y 359.87,Z 1042.829,A -85,B 0,C 180,E1 19834.151,E2 19834.151} C_VEL
LIN {X 0,Y 341.986,Z 980.778,A -85,B 0,C 180,E1 19837.912,E2 19837.912} C_VEL
LIN {X 0,Y 341.218,Z 977.53,A -85,B 0,C 180,E1 19838.196,E2 19838.196} C_VEL
LIN {X 0,Y 340.912,Z 977.53,A -85,B 0,C 180,E1 19845.348,E2 19845.348} C_VEL
LIN {X 0,Y 340.95,Z 977.53,A -85,B 0,C 180,E1 19853.148,E2 19853.148} C_VEL
LIN {X 0,Y 341.333,Z 977.53,A -85,B 0,C 180,E1 19860.756,E2 19860.756} C_VEL
LIN {X 0,Y 341.763,Z 977.53,A -85,B 0,C 180,E1 19868.635,E2 19868.635} C_VEL
LIN {X 0,Y 342.145,Z 977.53,A -85,B 0,C 180,E1 19874.578,E2 19874.578} C_VEL
LIN {X 0,Y 342.804,Z 977.53,A -85,B 0,C 180,E1 19882.368,E2 19882.368} C_VEL
LIN {X 0,Y 343.486,Z 977.53,A -85,B 0,C 180,E1 19889.988,E2 19889.988} C_VEL
LIN {X 0,Y 342.753,Z 977.53,A -85,B 0,C 180,E1 19897.609,E2 19897.609} C_VEL
LIN {X 0,Y 342.13,Z 977.53,A -85,B 0,C 180,E1 19905.398,E2 19905.398} C_VEL
LIN {X 0,Y 341.655,Z 977.53,A -85,B 0,C 180,E1 19913.513,E2 19913.513} C_VEL
LIN {X 0,Y 341.329,Z 977.53,A -85,B 0,C 180,E1 19919.217,E2 19919.217} C_VEL
LIN {X 0,Y 341.009,Z 977.53,A -85,B 0,C 180,E1 19926.865,E2 19926.865} C_VEL
LIN {X 0,Y 341.065,Z 978.296,A -85,B 0,C 180,E1 19933.32,E2 19933.32} C_VEL
LIN {X 0,Y 363.441,Z 1034.884,A -85,B 0,C 180,E1 19937.607,E2 19937.607} C_VEL
LIN {X 0,Y 376.338,Z 1075.295,A -85,B 0,C 180,E1 19941.019,E2 19941.019} C_VEL
LIN {X 0,Y 377.156,Z 1082.565,A -85,B 0,C 180,E1 19941.601,E2 19941.601} C_VEL
LIN {X 0,Y 370.12,Z 1122.512,A -85,B 0,C 180,E1 19944.655,E2 19944.655} C_VEL
LIN {X 0,Y 363.011,Z 1157.542,A -85,B 0,C 180,E1 19948.405,E2 19948.405} C_VEL
LIN {X 0,Y 356.284,Z 1188.488,A -85,B 0,C 180,E1 19952.896,E2 19952.896} C_VEL
LIN {X 0,Y 350.655,Z 1215.136,A -85,B 0,C 180,E1 19958.137,E2 19958.137} C_VEL
LIN {X 0,Y 346.706,Z 1236.597,A -85,B 0,C 180,E1 19964.007,E2 19964.007} C_VEL
LIN {X 0,Y 344.681,Z 1251.506,A -85,B 0,C 180,E1 19969.855,E2 19969.855} C_VEL
LIN {X 0,Y 343.911,Z 1260.059,A -85,B 0,C 180,E1 19974.927,E2 19974.927} C_VEL
LIN {X 0,Y 343.944,Z 1264.903,A -85,B 0,C 180,E1 19979.982,E2 19979.982} C_VEL
LIN {X 0,Y 344.318,Z 1266.341,A -85,B 0,C 180,E1 19985.031,E2 19985.031} C_VEL
LIN {X 0,Y 346.231,Z 1263.545,A -85,B 0,C 180,E1 19991.338,E2 19991.338} C_VEL
LIN {X 0,Y 350.855,Z 1254.784,A -85,B 0,C 180,E1 19998.208,E2 19998.208} C_VEL
LIN {X 0,Y 359.449,Z 1239.661,A -85,B 0,C 180,E1 20004.91,E2 20004.91} C_VEL
LIN {X 0,Y 371.44,Z 1219.472,A -85,B 0,C 180,E1 20010.825,E2 20010.825} C_VEL
LIN {X 0,Y 387.623,Z 1192.927,A -85,B 0,C 180,E1 20016.267,E2 20016.267} C_VEL
LIN {X 0,Y 407.375,Z 1160.599,A -85,B 0,C 180,E1 20020.937,E2 20020.937} C_VEL
LIN {X 0,Y 425.979,Z 1130.211,A -85,B 0,C 180,E1 20024.08,E2 20024.08} C_VEL
LIN {X 0,Y 426.422,Z 1129.523,A -85,B 0,C 180,E1 20024.329,E2 20024.329} C_VEL
LIN {X 0,Y 405.07,Z 1166.131,A -85,B 0,C 180,E1 20027.507,E2 20027.507} C_VEL
LIN {X 0,Y 383.756,Z 1204.055,A -85,B 0,C 180,E1 20032.289,E2 20032.289} C_VEL
LIN {X 0,Y 367.048,Z 1235.713,A -85,B 0,C 180,E1 20037.979,E2 20037.979} C_VEL
LIN {X 0,Y 355.228,Z 1260.457,A -85,B 0,C 180,E1 20044.232,E2 20044.232} C_VEL
LIN {X 0,Y 347.965,Z 1278.836,A -85,B 0,C 180,E1 20050.95,E2 20050.95} C_VEL
LIN {X 0,Y 344.752,Z 1290.069,A -85,B 0,C 180,E1 20057.317,E2 20057.317} C_VEL
LIN {X 0,Y 343.983,Z 1295.152,A -85,B 0,C 180,E1 20062.418,E2 20062.418} C_VEL
LIN {X 0,Y 343.916,Z 1296.739,A -85,B 0,C 180,E1 20067.487,E2 20067.487} C_VEL
LIN {X 0,Y 344.069,Z 1294.715,A -85,B 0,C 180,E1 20072.536,E2 20072.536} C_VEL
LIN {X 0,Y 344.245,Z 1287.105,A -85,B 0,C 180,E1 20078.578,E2 20078.578} C_VEL
LIN {X 0,Y 345.306,Z 1273.541,A -85,B 0,C 180,E1 20084.627,E2 20084.627} C_VEL
LIN {X 0,Y 353.155,Z 1237.614,A -85,B 0,C 180,E1 20095.76,E2 20095.76} C_VEL
LIN {X 0,Y 361.941,Z 1212.359,A -85,B 0,C 180,E1 20101.336,E2 20101.336} C_VEL
LIN {X 0,Y 373.474,Z 1181.138,A -85,B 0,C 180,E1 20106.301,E2 20106.301} C_VEL
LIN {X 0,Y 386.148,Z 1146.268,A -85,B 0,C 180,E1 20110.262,E2 20110.262} C_VEL
LIN {X 0,Y 400.083,Z 1104.799,A -85,B 0,C 180,E1 20113.549,E2 20113.549} C_VEL
LIN {X 0,Y 403.347,Z 1092.835,A -85,B 0,C 180,E1 20114.381,E2 20114.381} C_VEL
LIN {X 0,Y 403.491,Z 1081.798,A -85,B 0,C 180,E1 20115.823,E2 20115.823} C_VEL
LIN {X 0,Y 402.217,Z 1072.012,A -85,B 0,C 180,E1 20117.629,E2 20117.629} C_VEL
LIN {X 0,Y 399.68,Z 1067.602,A -85,B 0,C 180,E1 20119.358,E2 20119.358} C_VEL
LIN {X 0,Y 394.964,Z 1064.73,A -85,B 0,C 180,E1 20122.506,E2 20122.506} C_VEL
LIN {X 0,Y 393.805,Z 1061.992,A -85,B 0,C 180,E1 20124.773,E2 20124.773} C_VEL
LIN {X 0,Y 393.027,Z 1062.132,A -85,B 0,C 180,E1 20128.034,E2 20128.034} C_VEL
LIN {X 0,Y 393.63,Z 1065.844,A -85,B 0,C 180,E1 20131.148,E2 20131.148} C_VEL
LIN {X 0,Y 395.612,Z 1075.487,A -85,B 0,C 180,E1 20134.774,E2 20134.774} C_VEL
LIN {X 0,Y 396.805,Z 1084.945,A -85,B 0,C 180,E1 20136.894,E2 20136.894} C_VEL
LIN {X 0,Y 385.634,Z 1120.886,A -85,B 0,C 180,E1 20139.46,E2 20139.46} C_VEL
LIN {X 0,Y 375.332,Z 1148.078,A -85,B 0,C 180,E1 20142.473,E2 20142.473} C_VEL
LIN {X 0,Y 364.997,Z 1170.705,A -85,B 0,C 180,E1 20146.209,E2 20146.209} C_VEL
LIN {X 0,Y 356.274,Z 1186.96,A -85,B 0,C 180,E1 20150.224,E2 20150.224} C_VEL
LIN {X 0,Y 348.709,Z 1199.107,A -85,B 0,C 180,E1 20155.033,E2 20155.033} C_VEL
LIN {X 0,Y 343.205,Z 1205.735,A -85,B 0,C 180,E1 20160.018,E2 20160.018} C_VEL
LIN {X 0,Y 339.745,Z 1207.043,A -85,B 0,C 180,E1 20165.135,E2 20165.135} C_VEL
LIN {X 0,Y 338.328,Z 1203.015,A -85,B 0,C 180,E1 20170.337,E2 20170.337} C_VEL
LIN {X 0,Y 338.554,Z 1193.134,A -85,B 0,C 180,E1 20175.595,E2 20175.595} C_VEL
LIN {X 0,Y 340.044,Z 1177.818,A -85,B 0,C 180,E1 20180.477,E2 20180.477} C_VEL
LIN {X 0,Y 342.644,Z 1156.662,A -85,B 0,C 180,E1 20184.952,E2 20184.952} C_VEL
LIN {X 0,Y 345.704,Z 1132.366,A -85,B 0,C 180,E1 20188.484,E2 20188.484} C_VEL
LIN {X 0,Y 349.059,Z 1102.574,A -85,B 0,C 180,E1 20191.411,E2 20191.411} C_VEL
LIN {X 0,Y 351.499,Z 1070.101,A -85,B 0,C 180,E1 20193.375,E2 20193.375} C_VEL
LIN {X 0,Y 352.419,Z 1044.641,A -85,B 0,C 180,E1 20194.477,E2 20194.477} C_VEL
LIN {X 0,Y 335.012,Z 983.848,A -85,B 0,C 180,E1 20198.276,E2 20198.276} C_VEL
LIN {X 0,Y 333.228,Z 977.53,A -85,B 0,C 180,E1 20198.708,E2 20198.708} C_VEL
LIN {X 0,Y 332.899,Z 977.53,A -85,B 0,C 180,E1 20206.924,E2 20206.924} C_VEL
LIN {X 0,Y 333.045,Z 977.53,A -85,B 0,C 180,E1 20213.724,E2 20213.724} C_VEL
LIN {X 0,Y 333.29,Z 977.53,A -85,B 0,C 180,E1 20219.979,E2 20219.979} C_VEL
LIN {X 0,Y 333.673,Z 977.53,A -85,B 0,C 180,E1 20225.863,E2 20225.863} C_VEL
LIN {X 0,Y 334.107,Z 977.53,A -85,B 0,C 180,E1 20232.291,E2 20232.291} C_VEL
LIN {X 0,Y 334.586,Z 977.53,A -85,B 0,C 180,E1 20239.551,E2 20239.551} C_VEL
LIN {X 0,Y 335.304,Z 977.53,A -85,B 0,C 180,E1 20247.398,E2 20247.398} C_VEL
LIN {X 0,Y 335.32,Z 977.53,A -85,B 0,C 180,E1 20252.578,E2 20252.578} C_VEL
LIN {X 0,Y 334.569,Z 977.53,A -85,B 0,C 180,E1 20260.425,E2 20260.425} C_VEL
LIN {X 0,Y 334.008,Z 977.53,A -85,B 0,C 180,E1 20268.503,E2 20268.503} C_VEL
LIN {X 0,Y 333.591,Z 977.53,A -85,B 0,C 180,E1 20274.677,E2 20274.677} C_VEL
LIN {X 0,Y 333.172,Z 977.53,A -85,B 0,C 180,E1 20283.062,E2 20283.062} C_VEL
LIN {X 0,Y 333.097,Z 977.53,A -85,B 0,C 180,E1 20290.764,E2 20290.764} C_VEL
LIN {X 0,Y 333.133,Z 978.257,A -85,B 0,C 180,E1 20292.502,E2 20292.502} C_VEL
LIN {X 0,Y 355.815,Z 1035.438,A -85,B 0,C 180,E1 20296.99,E2 20296.99} C_VEL
LIN {X 0,Y 368.752,Z 1076.33,A -85,B 0,C 180,E1 20300.541,E2 20300.541} C_VEL
LIN {X 0,Y 369.906,Z 1083.149,A -85,B 0,C 180,E1 20301.129,E2 20301.129} C_VEL
LIN {X 0,Y 362.516,Z 1123.881,A -85,B 0,C 180,E1 20304.319,E2 20304.319} C_VEL
LIN {X 0,Y 355.185,Z 1159.227,A -85,B 0,C 180,E1 20308.211,E2 20308.211} C_VEL
LIN {X 0,Y 348.33,Z 1190.275,A -85,B 0,C 180,E1 20312.862,E2 20312.862} C_VEL
LIN {X 0,Y 342.527,Z 1217.163,A -85,B 0,C 180,E1 20318.374,E2 20318.374} C_VEL
LIN {X 0,Y 338.771,Z 1237.145,A -85,B 0,C 180,E1 20324.019,E2 20324.019} C_VEL
LIN {X 0,Y 336.696,Z 1252.542,A -85,B 0,C 180,E1 20330.266,E2 20330.266} C_VEL
LIN {X 0,Y 335.995,Z 1261.649,A -85,B 0,C 180,E1 20336.103,E2 20336.103} C_VEL
LIN {X 0,Y 336.047,Z 1265.173,A -85,B 0,C 180,E1 20339.982,E2 20339.982} C_VEL
LIN {X 0,Y 336.446,Z 1266.821,A -85,B 0,C 180,E1 20345.149,E2 20345.149} C_VEL
LIN {X 0,Y 337.964,Z 1265.279,A -85,B 0,C 180,E1 20350.311,E2 20350.311} C_VEL
LIN {X 0,Y 341.71,Z 1258.883,A -85,B 0,C 180,E1 20356.731,E2 20356.731} C_VEL
LIN {X 0,Y 349.66,Z 1246.101,A -85,B 0,C 180,E1 20363.609,E2 20363.609} C_VEL
LIN {X 0,Y 361.961,Z 1226.88,A -85,B 0,C 180,E1 20370.132,E2 20370.132} C_VEL
LIN {X 0,Y 378.242,Z 1202.291,A -85,B 0,C 180,E1 20375.841,E2 20375.841} C_VEL
LIN {X 0,Y 398.964,Z 1171.177,A -85,B 0,C 180,E1 20380.905,E2 20380.905} C_VEL
LIN {X 0,Y 416.969,Z 1144.521,A -85,B 0,C 180,E1 20384,E2 20384} C_VEL
LIN {X 0,Y 416.695,Z 1145.024,A -85,B 0,C 180,E1 20384.33,E2 20384.33} C_VEL
LIN {X 0,Y 392.476,Z 1183.24,A -85,B 0,C 180,E1 20388.256,E2 20388.256} C_VEL
LIN {X 0,Y 372.58,Z 1216.239,A -85,B 0,C 180,E1 20393.153,E2 20393.153} C_VEL
LIN {X 0,Y 356.744,Z 1244.583,A -85,B 0,C 180,E1 20399.015,E2 20399.015} C_VEL
LIN {X 0,Y 345.798,Z 1266.535,A -85,B 0,C 180,E1 20405.413,E2 20405.413} C_VEL
LIN {X 0,Y 339.048,Z 1282.962,A -85,B 0,C 180,E1 20412.455,E2 20412.455} C_VEL
LIN {X 0,Y 336.403,Z 1292.856,A -85,B 0,C 180,E1 20419.632,E2 20419.632} C_VEL
LIN {X 0,Y 335.941,Z 1295.998,A -85,B 0,C 180,E1 20424.836,E2 20424.836} C_VEL
LIN {X 0,Y 336.29,Z 1295.652,A -85,B 0,C 180,E1 20430.012,E2 20430.012} C_VEL
LIN {X 0,Y 336.229,Z 1291.371,A -85,B 0,C 180,E1 20435.183,E2 20435.183} C_VEL
LIN {X 0,Y 336.603,Z 1281.756,A -85,B 0,C 180,E1 20441.042,E2 20441.042} C_VEL
LIN {X 0,Y 338.206,Z 1266.413,A -85,B 0,C 180,E1 20446.943,E2 20446.943} C_VEL
LIN {X 0,Y 345.927,Z 1237.624,A -85,B 0,C 180,E1 20456.339,E2 20456.339} C_VEL
LIN {X 0,Y 355.548,Z 1211.827,A -85,B 0,C 180,E1 20462.203,E2 20462.203} C_VEL
LIN {X 0,Y 368.251,Z 1179.768,A -85,B 0,C 180,E1 20467.381,E2 20467.381} C_VEL
LIN {X 0,Y 381.884,Z 1144.264,A -85,B 0,C 180,E1 20471.416,E2 20471.416} C_VEL
LIN {X 0,Y 396.397,Z 1103.37,A -85,B 0,C 180,E1 20474.629,E2 20474.629} C_VEL
LIN {X 0,Y 398.797,Z 1094.363,A -85,B 0,C 180,E1 20475.331,E2 20475.331} C_VEL
LIN {X 0,Y 398.558,Z 1081.382,A -85,B 0,C 180,E1 20477.373,E2 20477.373} C_VEL
LIN {X 0,Y 396.631,Z 1069.4,A -85,B 0,C 180,E1 20480.338,E2 20480.338} C_VEL
LIN {X 0,Y 394.964,Z 1064.73,A -85,B 0,C 180,E1 20482.506,E2 20482.506} C_VEL
LIN {X 0,Y 392.933,Z 1064.742,A -85,B 0,C 180,E1 20484.382,E2 20484.382} C_VEL
LIN {X 0,Y 389.908,Z 1069.185,A -85,B 0,C 180,E1 20487.551,E2 20487.551} C_VEL
LIN {X 0,Y 390.355,Z 1073.59,A -85,B 0,C 180,E1 20491.335,E2 20491.335} C_VEL
LIN {X 0,Y 391.936,Z 1083.521,A -85,B 0,C 180,E1 20494.853,E2 20494.853} C_VEL
LIN {X 0,Y 392.559,Z 1088.297,A -85,B 0,C 180,E1 20496.02,E2 20496.02} C_VEL
LIN {X 0,Y 380.873,Z 1123.09,A -85,B 0,C 180,E1 20498.581,E2 20498.581} C_VEL
LIN {X 0,Y 370.309,Z 1149.229,A -85,B 0,C 180,E1 20501.531,E2 20501.531} C_VEL
LIN {X 0,Y 359.194,Z 1172.001,A -85,B 0,C 180,E1 20505.358,E2 20505.358} C_VEL
LIN {X 0,Y 349.935,Z 1188.158,A -85,B 0,C 180,E1 20509.415,E2 20509.415} C_VEL
LIN {X 0,Y 342.047,Z 1199.948,A -85,B 0,C 180,E1 20514.147,E2 20514.147} C_VEL
LIN {X 0,Y 336.537,Z 1206.262,A -85,B 0,C 180,E1 20518.729,E2 20518.729} C_VEL
LIN {X 0,Y 333.327,Z 1208.278,A -85,B 0,C 180,E1 20522.624,E2 20522.624} C_VEL
LIN {X 0,Y 330.902,Z 1206.382,A -85,B 0,C 180,E1 20527.914,E2 20527.914} C_VEL
LIN {X 0,Y 330.422,Z 1198.896,A -85,B 0,C 180,E1 20533.273,E2 20533.273} C_VEL
LIN {X 0,Y 331.33,Z 1186.156,A -85,B 0,C 180,E1 20538.343,E2 20538.343} C_VEL
LIN {X 0,Y 333.419,Z 1167.66,A -85,B 0,C 180,E1 20543.095,E2 20543.095} C_VEL
LIN {X 0,Y 336.527,Z 1144.834,A -85,B 0,C 180,E1 20547.125,E2 20547.125} C_VEL
LIN {X 0,Y 339.847,Z 1117.065,A -85,B 0,C 180,E1 20550.493,E2 20550.493} C_VEL
LIN {X 0,Y 342.873,Z 1086.752,A -85,B 0,C 180,E1 20552.873,E2 20552.873} C_VEL
LIN {X 0,Y 344.826,Z 1045.906,A -85,B 0,C 180,E1 20554.841,E2 20554.841} C_VEL
LIN {X 0,Y 328.062,Z 986.937,A -85,B 0,C 180,E1 20558.651,E2 20558.651} C_VEL
LIN {X 0,Y 325.255,Z 977.53,A -85,B 0,C 180,E1 20559.41,E2 20559.41} C_VEL
LIN {X 0,Y 324.901,Z 977.53,A -85,B 0,C 180,E1 20568.284,E2 20568.284} C_VEL
LIN {X 0,Y 325.195,Z 977.53,A -85,B 0,C 180,E1 20575.988,E2 20575.988} C_VEL
LIN {X 0,Y 325.49,Z 977.53,A -85,B 0,C 180,E1 20582.241,E2 20582.241} C_VEL
LIN {X 0,Y 325.949,Z 977.53,A -85,B 0,C 180,E1 20588.431,E2 20588.431} C_VEL
LIN {X 0,Y 326.476,Z 977.53,A -85,B 0,C 180,E1 20596.569,E2 20596.569} C_VEL
LIN {X 0,Y 327.203,Z 977.53,A -85,B 0,C 180,E1 20604.673,E2 20604.673} C_VEL
LIN {X 0,Y 327.675,Z 977.53,A -85,B 0,C 180,E1 20609.988,E2 20609.988} C_VEL
LIN {X 0,Y 326.878,Z 977.53,A -85,B 0,C 180,E1 20617.981,E2 20617.981} C_VEL
LIN {X 0,Y 326.46,Z 977.53,A -85,B 0,C 180,E1 20623.407,E2 20623.407} C_VEL
LIN {X 0,Y 325.861,Z 977.53,A -85,B 0,C 180,E1 20631.826,E2 20631.826} C_VEL
LIN {X 0,Y 325.483,Z 977.53,A -85,B 0,C 180,E1 20637.778,E2 20637.778} C_VEL
LIN {X 0,Y 325.249,Z 977.53,A -85,B 0,C 180,E1 20643.975,E2 20643.975} C_VEL
LIN {X 0,Y 325.216,Z 978.228,A -85,B 0,C 180,E1 20651.675,E2 20651.675} C_VEL
LIN {X 0,Y 347.487,Z 1034.325,A -85,B 0,C 180,E1 20656.222,E2 20656.222} C_VEL
LIN {X 0,Y 360.712,Z 1075.645,A -85,B 0,C 180,E1 20659.886,E2 20659.886} C_VEL
LIN {X 0,Y 362.426,Z 1085.056,A -85,B 0,C 180,E1 20660.723,E2 20660.723} C_VEL
LIN {X 0,Y 354.968,Z 1125.128,A -85,B 0,C 180,E1 20663.965,E2 20663.965} C_VEL
LIN {X 0,Y 347.524,Z 1160.052,A -85,B 0,C 180,E1 20667.905,E2 20667.905} C_VEL
LIN {X 0,Y 340.381,Z 1191.719,A -85,B 0,C 180,E1 20672.78,E2 20672.78} C_VEL
LIN {X 0,Y 334.498,Z 1218.47,A -85,B 0,C 180,E1 20678.456,E2 20678.456} C_VEL
LIN {X 0,Y 330.845,Z 1237.756,A -85,B 0,C 180,E1 20684.067,E2 20684.067} C_VEL
LIN {X 0,Y 328.862,Z 1252.277,A -85,B 0,C 180,E1 20690.032,E2 20690.032} C_VEL
LIN {X 0,Y 328.094,Z 1261.706,A -85,B 0,C 180,E1 20696.009,E2 20696.009} C_VEL
LIN {X 0,Y 328.161,Z 1265.403,A -85,B 0,C 180,E1 20699.981,E2 20699.981} C_VEL
LIN {X 0,Y 328.575,Z 1267.303,A -85,B 0,C 180,E1 20705.272,E2 20705.272} C_VEL
LIN {X 0,Y 330.186,Z 1266.001,A -85,B 0,C 180,E1 20710.557,E2 20710.557} C_VEL
LIN {X 0,Y 334.194,Z 1260.002,A -85,B 0,C 180,E1 20717.119,E2 20717.119} C_VEL
LIN {X 0,Y 342.448,Z 1247.963,A -85,B 0,C 180,E1 20724.037,E2 20724.037} C_VEL
LIN {X 0,Y 355.506,Z 1229.397,A -85,B 0,C 180,E1 20730.738,E2 20730.738} C_VEL
LIN {X 0,Y 372.473,Z 1205.832,A -85,B 0,C 180,E1 20736.484,E2 20736.484} C_VEL
LIN {X 0,Y 395.147,Z 1174.853,A -85,B 0,C 180,E1 20741.753,E2 20741.753} C_VEL
LIN {X 0,Y 408.029,Z 1157.472,A -85,B 0,C 180,E1 20743.922,E2 20743.922} C_VEL
LIN {X 0,Y 408.395,Z 1156.985,A -85,B 0,C 180,E1 20744.166,E2 20744.166} C_VEL
LIN {X 0,Y 383.805,Z 1192.653,A -85,B 0,C 180,E1 20748.238,E2 20748.238} C_VEL
LIN {X 0,Y 363.112,Z 1224.561,A -85,B 0,C 180,E1 20753.526,E2 20753.526} C_VEL
LIN {X 0,Y 347.594,Z 1250.569,A -85,B 0,C 180,E1 20759.565,E2 20759.565} C_VEL
LIN {X 0,Y 336.968,Z 1270.61,A -85,B 0,C 180,E1 20766.14,E2 20766.14} C_VEL
LIN {X 0,Y 330.6,Z 1285.357,A -85,B 0,C 180,E1 20773.367,E2 20773.367} C_VEL
LIN {X 0,Y 328.531,Z 1292.668,A -85,B 0,C 180,E1 20779.381,E2 20779.381} C_VEL
LIN {X 0,Y 328.061,Z 1295.619,A -85,B 0,C 180,E1 20784.712,E2 20784.712} C_VEL
LIN {X 0,Y 328.418,Z 1295.036,A -85,B 0,C 180,E1 20790.012,E2 20790.012} C_VEL
LIN {X 0,Y 328.407,Z 1289.112,A -85,B 0,C 180,E1 20796.453,E2 20796.453} C_VEL
LIN {X 0,Y 329.003,Z 1277.73,A -85,B 0,C 180,E1 20802.649,E2 20802.649} C_VEL
LIN {X 0,Y 332.843,Z 1254.636,A -85,B 0,C 180,E1 20811.371,E2 20811.371} C_VEL
LIN {X 0,Y 340.016,Z 1234.077,A -85,B 0,C 180,E1 20817.913,E2 20817.913} C_VEL
LIN {X 0,Y 350.849,Z 1207.714,A -85,B 0,C 180,E1 20823.797,E2 20823.797} C_VEL
LIN {X 0,Y 363.844,Z 1177.149,A -85,B 0,C 180,E1 20828.673,E2 20828.673} C_VEL
LIN {X 0,Y 378.198,Z 1141.751,A -85,B 0,C 180,E1 20832.653,E2 20832.653} C_VEL
LIN {X 0,Y 394.1,Z 1097.877,A -85,B 0,C 180,E1 20836.096,E2 20836.096} C_VEL
LIN {X 0,Y 394.119,Z 1084.791,A -85,B 0,C 180,E1 20838.34,E2 20838.34} C_VEL
LIN {X 0,Y 392.76,Z 1075.292,A -85,B 0,C 180,E1 20840.961,E2 20840.961} C_VEL
LIN {X 0,Y 390.695,Z 1069.519,A -85,B 0,C 180,E1 20844.552,E2 20844.552} C_VEL
LIN {X 0,Y 389.908,Z 1069.185,A -85,B 0,C 180,E1 20847.551,E2 20847.551} C_VEL
LIN {X 0,Y 388.864,Z 1073.068,A -85,B 0,C 180,E1 20849.391,E2 20849.391} C_VEL
LIN {X 0,Y 387.207,Z 1083.201,A -85,B 0,C 180,E1 20852.322,E2 20852.322} C_VEL
LIN {X 0,Y 388.173,Z 1091.99,A -85,B 0,C 180,E1 20855.046,E2 20855.046} C_VEL
LIN {X 0,Y 374.771,Z 1129.347,A -85,B 0,C 180,E1 20858.058,E2 20858.058} C_VEL
LIN {X 0,Y 363.397,Z 1154.69,A -85,B 0,C 180,E1 20861.167,E2 20861.167} C_VEL
LIN {X 0,Y 351.193,Z 1177.333,A -85,B 0,C 180,E1 20865.336,E2 20865.336} C_VEL
LIN {X 0,Y 341.333,Z 1192.941,A -85,B 0,C 180,E1 20869.791,E2 20869.791} C_VEL
LIN {X 0,Y 333.269,Z 1203.491,A -85,B 0,C 180,E1 20874.802,E2 20874.802} C_VEL
LIN {X 0,Y 327.494,Z 1208.764,A -85,B 0,C 180,E1 20880.019,E2 20880.019} C_VEL
LIN {X 0,Y 323.935,Z 1208.859,A -85,B 0,C 180,E1 20885.387,E2 20885.387} C_VEL
LIN {X 0,Y 322.558,Z 1203.631,A -85,B 0,C 180,E1 20890.849,E2 20890.849} C_VEL
LIN {X 0,Y 322.934,Z 1192.493,A -85,B 0,C 180,E1 20896.37,E2 20896.37} C_VEL
LIN {X 0,Y 324.797,Z 1175.4,A -85,B 0,C 180,E1 20901.585,E2 20901.585} C_VEL
LIN {X 0,Y 327.693,Z 1152.649,A -85,B 0,C 180,E1 20906.193,E2 20906.193} C_VEL
LIN {X 0,Y 331.038,Z 1127.05,A -85,B 0,C 180,E1 20909.752,E2 20909.752} C_VEL
LIN {X 0,Y 334.445,Z 1096.928,A -85,B 0,C 180,E1 20912.567,E2 20912.567} C_VEL
LIN {X 0,Y 336.978,Z 1062.539,A -85,B 0,C 180,E1 20914.496,E2 20914.496} C_VEL
LIN {X 0,Y 337.174,Z 1046.817,A -85,B 0,C 180,E1 20915.238,E2 20915.238} C_VEL
LIN {X 0,Y 320.524,Z 988.166,A -85,B 0,C 180,E1 20919.148,E2 20919.148} C_VEL
LIN {X 0,Y 317.224,Z 977.53,A -85,B 0,C 180,E1 20920.043,E2 20920.043} C_VEL
LIN {X 0,Y 316.98,Z 977.53,A -85,B 0,C 180,E1 20927.974,E2 20927.974} C_VEL
LIN {X 0,Y 317.127,Z 977.53,A -85,B 0,C 180,E1 20934.999,E2 20934.999} C_VEL
LIN {X 0,Y 317.478,Z 977.53,A -85,B 0,C 180,E1 20941.478,E2 20941.478} C_VEL
LIN {X 0,Y 317.887,Z 977.53,A -85,B 0,C 180,E1 20947.57,E2 20947.57} C_VEL
LIN {X 0,Y 318.284,Z 977.53,A -85,B 0,C 180,E1 20953.389,E2 20953.389} C_VEL
LIN {X 0,Y 318.986,Z 977.53,A -85,B 0,C 180,E1 20961.794,E2 20961.794} C_VEL
LIN {X 0,Y 319.77,Z 977.53,A -85,B 0,C 180,E1 20969.987,E2 20969.987} C_VEL
LIN {X 0,Y 318.949,Z 977.53,A -85,B 0,C 180,E1 20978.181,E2 20978.181} C_VEL
LIN {X 0,Y 318.258,Z 977.53,A -85,B 0,C 180,E1 20986.585,E2 20986.585} C_VEL
LIN {X 0,Y 317.751,Z 977.53,A -85,B 0,C 180,E1 20995.003,E2 20995.003} C_VEL
LIN {X 0,Y 317.363,Z 977.53,A -85,B 0,C 180,E1 21001.667,E2 21001.667} C_VEL
LIN {X 0,Y 317.32,Z 977.587,A -85,B 0,C 180,E1 21010.789,E2 21010.789} C_VEL
LIN {X 0,Y 340.224,Z 1035.951,A -85,B 0,C 180,E1 21015.657,E2 21015.657} C_VEL
LIN {X 0,Y 353.219,Z 1077.079,A -85,B 0,C 180,E1 21019.418,E2 21019.418} C_VEL
LIN {X 0,Y 355.001,Z 1086.639,A -85,B 0,C 180,E1 21020.302,E2 21020.302} C_VEL
LIN {X 0,Y 347.434,Z 1126.069,A -85,B 0,C 180,E1 21023.573,E2 21023.573} C_VEL
LIN {X 0,Y 339.799,Z 1161.159,A -85,B 0,C 180,E1 21027.631,E2 21027.631} C_VEL
LIN {X 0,Y 332.543,Z 1192.509,A -85,B 0,C 180,E1 21032.588,E2 21032.588} C_VEL
LIN {X 0,Y 326.726,Z 1218.435,A -85,B 0,C 180,E1 21038.204,E2 21038.204} C_VEL
LIN {X 0,Y 322.767,Z 1239.099,A -85,B 0,C 180,E1 21044.392,E2 21044.392} C_VEL
LIN {X 0,Y 320.877,Z 1253.268,A -85,B 0,C 180,E1 21050.468,E2 21050.468} C_VEL
LIN {X 0,Y 320.205,Z 1261.719,A -85,B 0,C 180,E1 21055.911,E2 21055.911} C_VEL
LIN {X 0,Y 320.394,Z 1267.116,A -85,B 0,C 180,E1 21062.691,E2 21062.691} C_VEL
LIN {X 0,Y 321.463,Z 1267.611,A -85,B 0,C 180,E1 21068.253,E2 21068.253} C_VEL
LIN {X 0,Y 325.606,Z 1262.678,A -85,B 0,C 180,E1 21076.192,E2 21076.192} C_VEL
LIN {X 0,Y 333.627,Z 1252.101,A -85,B 0,C 180,E1 21083.393,E2 21083.393} C_VEL
LIN {X 0,Y 346.276,Z 1235.559,A -85,B 0,C 180,E1 21090.189,E2 21090.189} C_VEL
LIN {X 0,Y 364.867,Z 1211.9,A -85,B 0,C 180,E1 21096.628,E2 21096.628} C_VEL
LIN {X 0,Y 389.128,Z 1181.531,A -85,B 0,C 180,E1 21102.172,E2 21102.172} C_VEL
LIN {X 0,Y 399.048,Z 1169.319,A -85,B 0,C 180,E1 21103.839,E2 21103.839} C_VEL
LIN {X 0,Y 398.084,Z 1170.629,A -85,B 0,C 180,E1 21104.257,E2 21104.257} C_VEL
LIN {X 0,Y 371.83,Z 1205.929,A -85,B 0,C 180,E1 21108.934,E2 21108.934} C_VEL
LIN {X 0,Y 349.454,Z 1238.476,A -85,B 0,C 180,E1 21115.326,E2 21115.326} C_VEL
LIN {X 0,Y 334.457,Z 1262.49,A -85,B 0,C 180,E1 21122.217,E2 21122.217} C_VEL
LIN {X 0,Y 325.366,Z 1279.782,A -85,B 0,C 180,E1 21129.57,E2 21129.57} C_VEL
LIN {X 0,Y 321.34,Z 1289.876,A -85,B 0,C 180,E1 21136.376,E2 21136.376} C_VEL
LIN {X 0,Y 320.165,Z 1294.903,A -85,B 0,C 180,E1 21143.425,E2 21143.425} C_VEL
LIN {X 0,Y 320.566,Z 1294.374,A -85,B 0,C 180,E1 21150.013,E2 21150.013} C_VEL
LIN {X 0,Y 320.482,Z 1289.684,A -85,B 0,C 180,E1 21155.439,E2 21155.439} C_VEL
LIN {X 0,Y 320.95,Z 1279.462,A -85,B 0,C 180,E1 21161.588,E2 21161.588} C_VEL
LIN {X 0,Y 323.703,Z 1259.532,A -85,B 0,C 180,E1 21169.652,E2 21169.652} C_VEL
LIN {X 0,Y 329.664,Z 1242.357,A -85,B 0,C 180,E1 21176.158,E2 21176.158} C_VEL
LIN {X 0,Y 339.626,Z 1218.818,A -85,B 0,C 180,E1 21182.384,E2 21182.384} C_VEL
LIN {X 0,Y 352.683,Z 1190.146,A -85,B 0,C 180,E1 21187.766,E2 21187.766} C_VEL
LIN {X 0,Y 368.028,Z 1155.742,A -85,B 0,C 180,E1 21192.277,E2 21192.277} C_VEL
LIN {X 0,Y 383.605,Z 1117.55,A -85,B 0,C 180,E1 21195.722,E2 21195.722} C_VEL
LIN {X 0,Y 389.665,Z 1100.642,A -85,B 0,C 180,E1 21196.979,E2 21196.979} C_VEL
LIN {X 0,Y 389.785,Z 1088.388,A -85,B 0,C 180,E1 21199.361,E2 21199.361} C_VEL
LIN {X 0,Y 388.93,Z 1081.494,A -85,B 0,C 180,E1 21201.464,E2 21201.464} C_VEL
LIN {X 0,Y 387.533,Z 1077.25,A -85,B 0,C 180,E1 21204.115,E2 21204.115} C_VEL
LIN {X 0,Y 386.646,Z 1076.542,A -85,B 0,C 180,E1 21207.44,E2 21207.44} C_VEL
LIN {X 0,Y 386.778,Z 1079.853,A -85,B 0,C 180,E1 21210.73,E2 21210.73} C_VEL
LIN {X 0,Y 387.207,Z 1083.201,A -85,B 0,C 180,E1 21212.322,E2 21212.322} C_VEL
LIN {X 0,Y 386.191,Z 1089.663,A -85,B 0,C 180,E1 21213.586,E2 21213.586} C_VEL
LIN {X 0,Y 381.73,Z 1102.938,A -85,B 0,C 180,E1 21214.727,E2 21214.727} C_VEL
LIN {X 0,Y 378.669,Z 1110.98,A -85,B 0,C 180,E1 21215.296,E2 21215.296} C_VEL
LIN {X 0,Y 366.676,Z 1139.619,A -85,B 0,C 180,E1 21217.992,E2 21217.992} C_VEL
LIN {X 0,Y 353.842,Z 1164.849,A -85,B 0,C 180,E1 21221.61,E2 21221.61} C_VEL
LIN {X 0,Y 341.716,Z 1184.621,A -85,B 0,C 180,E1 21225.904,E2 21225.904} C_VEL
LIN {X 0,Y 331.538,Z 1198.759,A -85,B 0,C 180,E1 21230.809,E2 21230.809} C_VEL
LIN {X 0,Y 323.843,Z 1207.216,A -85,B 0,C 180,E1 21235.995,E2 21235.995} C_VEL
LIN {X 0,Y 318.389,Z 1210.549,A -85,B 0,C 180,E1 21241.533,E2 21241.533} C_VEL
LIN {X 0,Y 315.483,Z 1208.736,A -85,B 0,C 180,E1 21246.915,E2 21246.915} C_VEL
LIN {X 0,Y 314.646,Z 1201.497,A -85,B 0,C 180,E1 21252.535,E2 21252.535} C_VEL
LIN {X 0,Y 315.509,Z 1188.017,A -85,B 0,C 180,E1 21258.208,E2 21258.208} C_VEL
LIN {X 0,Y 317.64,Z 1169.584,A -85,B 0,C 180,E1 21263.194,E2 21263.194} C_VEL
LIN {X 0,Y 320.856,Z 1146.548,A -85,B 0,C 180,E1 21267.468,E2 21267.468} C_VEL
LIN {X 0,Y 324.281,Z 1119.298,A -85,B 0,C 180,E1 21270.949,E2 21270.949} C_VEL
LIN {X 0,Y 327.59,Z 1088.633,A -85,B 0,C 180,E1 21273.515,E2 21273.515} C_VEL
LIN {X 0,Y 329.684,Z 1048.164,A -85,B 0,C 180,E1 21275.618,E2 21275.618} C_VEL
LIN {X 0,Y 312.982,Z 989.612,A -85,B 0,C 180,E1 21279.654,E2 21279.654} C_VEL
LIN {X 0,Y 309.26,Z 977.53,A -85,B 0,C 180,E1 21280.587,E2 21280.587} C_VEL
LIN {X 0,Y 309.061,Z 977.53,A -85,B 0,C 180,E1 21287.365,E2 21287.365} C_VEL
LIN {X 0,Y 309.128,Z 977.53,A -85,B 0,C 180,E1 21293.954,E2 21293.954} C_VEL
LIN {X 0,Y 309.582,Z 977.53,A -85,B 0,C 180,E1 21301.795,E2 21301.795} C_VEL
LIN {X 0,Y 310.102,Z 977.53,A -85,B 0,C 180,E1 21309.985,E2 21309.985} C_VEL
LIN {X 0,Y 310.612,Z 977.53,A -85,B 0,C 180,E1 21317.394,E2 21317.394} C_VEL
LIN {X 0,Y 311.341,Z 977.53,A -85,B 0,C 180,E1 21324.401,E2 21324.401} C_VEL
LIN {X 0,Y 311.883,Z 977.53,A -85,B 0,C 180,E1 21329.987,E2 21329.987} C_VEL
LIN {X 0,Y 311,Z 977.53,A -85,B 0,C 180,E1 21338.392,E2 21338.392} C_VEL
LIN {X 0,Y 310.531,Z 977.53,A -85,B 0,C 180,E1 21344.108,E2 21344.108} C_VEL
LIN {X 0,Y 309.944,Z 977.53,A -85,B 0,C 180,E1 21351.702,E2 21351.702} C_VEL
LIN {X 0,Y 309.515,Z 977.53,A -85,B 0,C 180,E1 21359.297,E2 21359.297} C_VEL
LIN {X 0,Y 309.194,Z 977.53,A -85,B 0,C 180,E1 21366.005,E2 21366.005} C_VEL
LIN {X 0,Y 309.308,Z 977.846,A -85,B 0,C 180,E1 21369.883,E2 21369.883} C_VEL
LIN {X 0,Y 332.089,Z 1035.296,A -85,B 0,C 180,E1 21374.878,E2 21374.878} C_VEL
LIN {X 0,Y 345.261,Z 1076.61,A -85,B 0,C 180,E1 21378.756,E2 21378.756} C_VEL
LIN {X 0,Y 347.466,Z 1088.594,A -85,B 0,C 180,E1 21379.898,E2 21379.898} C_VEL
LIN {X 0,Y 339.975,Z 1126.736,A -85,B 0,C 180,E1 21383.15,E2 21383.15} C_VEL
LIN {X 0,Y 332.06,Z 1162.231,A -85,B 0,C 180,E1 21387.355,E2 21387.355} C_VEL
LIN {X 0,Y 324.388,Z 1194.488,A -85,B 0,C 180,E1 21392.636,E2 21392.636} C_VEL
LIN {X 0,Y 318.68,Z 1219.937,A -85,B 0,C 180,E1 21398.359,E2 21398.359} C_VEL
LIN {X 0,Y 314.848,Z 1239.482,A -85,B 0,C 180,E1 21404.395,E2 21404.395} C_VEL
LIN {X 0,Y 312.9,Z 1254.235,A -85,B 0,C 180,E1 21410.926,E2 21410.926} C_VEL
LIN {X 0,Y 312.235,Z 1263.198,A -85,B 0,C 180,E1 21417.199,E2 21417.199} C_VEL
LIN {X 0,Y 312.498,Z 1267.376,A -85,B 0,C 180,E1 21422.759,E2 21422.759} C_VEL
LIN {X 0,Y 313.598,Z 1268.259,A -85,B 0,C 180,E1 21428.314,E2 21428.314} C_VEL
LIN {X 0,Y 318.051,Z 1263.724,A -85,B 0,C 180,E1 21436.587,E2 21436.587} C_VEL
LIN {X 0,Y 327.543,Z 1252.537,A -85,B 0,C 180,E1 21444.581,E2 21444.581} C_VEL
LIN {X 0,Y 342.738,Z 1234.491,A -85,B 0,C 180,E1 21452.015,E2 21452.015} C_VEL
LIN {X 0,Y 363.171,Z 1210.889,A -85,B 0,C 180,E1 21458.335,E2 21458.335} C_VEL
LIN {X 0,Y 387.952,Z 1182.558,A -85,B 0,C 180,E1 21463.475,E2 21463.475} C_VEL
LIN {X 0,Y 389.81,Z 1180.493,A -85,B 0,C 180,E1 21463.776,E2 21463.776} C_VEL
LIN {X 0,Y 388.112,Z 1182.605,A -85,B 0,C 180,E1 21464.306,E2 21464.306} C_VEL
LIN {X 0,Y 363.183,Z 1213.713,A -85,B 0,C 180,E1 21468.934,E2 21468.934} C_VEL
LIN {X 0,Y 340.927,Z 1243.704,A -85,B 0,C 180,E1 21475.425,E2 21475.425} C_VEL
LIN {X 0,Y 325.176,Z 1267.241,A -85,B 0,C 180,E1 21482.992,E2 21482.992} C_VEL
LIN {X 0,Y 316.696,Z 1282.494,A -85,B 0,C 180,E1 21490.446,E2 21490.446} C_VEL
LIN {X 0,Y 313.109,Z 1291.189,A -85,B 0,C 180,E1 21497.435,E2 21497.435} C_VEL
LIN {X 0,Y 312.282,Z 1294.806,A -85,B 0,C 180,E1 21504.444,E2 21504.444} C_VEL
LIN {X 0,Y 312.689,Z 1293.698,A -85,B 0,C 180,E1 21510.013,E2 21510.013} C_VEL
LIN {X 0,Y 312.706,Z 1287.609,A -85,B 0,C 180,E1 21516.486,E2 21516.486} C_VEL
LIN {X 0,Y 313.247,Z 1276.775,A -85,B 0,C 180,E1 21522.586,E2 21522.586} C_VEL
LIN {X 0,Y 315.078,Z 1262.874,A -85,B 0,C 180,E1 21528.229,E2 21528.229} C_VEL
LIN {X 0,Y 320.991,Z 1245.847,A -85,B 0,C 180,E1 21535.606,E2 21535.606} C_VEL
LIN {X 0,Y 331.038,Z 1223.389,A -85,B 0,C 180,E1 21542.177,E2 21542.177} C_VEL
LIN {X 0,Y 344.873,Z 1194.976,A -85,B 0,C 180,E1 21547.975,E2 21547.975} C_VEL
LIN {X 0,Y 360.666,Z 1162.17,A -85,B 0,C 180,E1 21552.629,E2 21552.629} C_VEL
LIN {X 0,Y 376.141,Z 1127.007,A -85,B 0,C 180,E1 21556.077,E2 21556.077} C_VEL
LIN {X 0,Y 385.271,Z 1103.58,A -85,B 0,C 180,E1 21557.908,E2 21557.908} C_VEL
LIN {X 0,Y 385.637,Z 1092.545,A -85,B 0,C 180,E1 21560.275,E2 21560.275} C_VEL
LIN {X 0,Y 384.68,Z 1086.021,A -85,B 0,C 180,E1 21562.871,E2 21562.871} C_VEL
LIN {X 0,Y 383.406,Z 1083.324,A -85,B 0,C 180,E1 21566.431,E2 21566.431} C_VEL
LIN {X 0,Y 383.171,Z 1084.707,A -85,B 0,C 180,E1 21569.086,E2 21569.086} C_VEL
LIN {X 0,Y 383.548,Z 1090.744,A -85,B 0,C 180,E1 21572.363,E2 21572.363} C_VEL
LIN {X 0,Y 383.945,Z 1096.84,A -85,B 0,C 180,E1 21574.292,E2 21574.292} C_VEL
LIN {X 0,Y 378.669,Z 1110.98,A -85,B 0,C 180,E1 21575.296,E2 21575.296} C_VEL
LIN {X 0,Y 370.992,Z 1126.311,A -85,B 0,C 180,E1 21575.992,E2 21575.992} C_VEL
LIN {X 0,Y 363.705,Z 1138.833,A -85,B 0,C 180,E1 21576.694,E2 21576.694} C_VEL
LIN {X 0,Y 362.87,Z 1140.446,A -85,B 0,C 180,E1 21576.869,E2 21576.869} C_VEL
LIN {X 0,Y 349.567,Z 1165.06,A -85,B 0,C 180,E1 21580.392,E2 21580.392} C_VEL
LIN {X 0,Y 335.942,Z 1186.095,A -85,B 0,C 180,E1 21584.989,E2 21584.989} C_VEL
LIN {X 0,Y 325.102,Z 1200.043,A -85,B 0,C 180,E1 21589.955,E2 21589.955} C_VEL
LIN {X 0,Y 316.058,Z 1209.083,A -85,B 0,C 180,E1 21595.896,E2 21595.896} C_VEL
LIN {X 0,Y 311.77,Z 1211.562,A -85,B 0,C 180,E1 21600.02,E2 21600.02} C_VEL
LIN {X 0,Y 308.11,Z 1210.41,A -85,B 0,C 180,E1 21605.664,E2 21605.664} C_VEL
LIN {X 0,Y 306.787,Z 1203.939,A -85,B 0,C 180,E1 21611.414,E2 21611.414} C_VEL
LIN {X 0,Y 307.219,Z 1192.931,A -85,B 0,C 180,E1 21616.691,E2 21616.691} C_VEL
LIN {X 0,Y 309.171,Z 1175.607,A -85,B 0,C 180,E1 21622.002,E2 21622.002} C_VEL
LIN {X 0,Y 312.158,Z 1153.091,A -85,B 0,C 180,E1 21626.699,E2 21626.699} C_VEL
LIN {X 0,Y 315.674,Z 1127.332,A -85,B 0,C 180,E1 21630.405,E2 21630.405} C_VEL
LIN {X 0,Y 319.2,Z 1097.458,A -85,B 0,C 180,E1 21633.278,E2 21633.278} C_VEL
LIN {X 0,Y 322.066,Z 1060.953,A -85,B 0,C 180,E1 21635.406,E2 21635.406} C_VEL
LIN {X 0,Y 321.749,Z 1048.174,A -85,B 0,C 180,E1 21636.089,E2 21636.089} C_VEL
LIN {X 0,Y 305.483,Z 991.004,A -85,B 0,C 180,E1 21640.186,E2 21640.186} C_VEL
LIN {X 0,Y 301.291,Z 977.53,A -85,B 0,C 180,E1 21641.406,E2 21641.406} C_VEL
LIN {X 0,Y 301.054,Z 977.53,A -85,B 0,C 180,E1 21649.115,E2 21649.115} C_VEL
LIN {X 0,Y 301.286,Z 977.53,A -85,B 0,C 180,E1 21656.395,E2 21656.395} C_VEL
LIN {X 0,Y 301.789,Z 977.53,A -85,B 0,C 180,E1 21664.692,E2 21664.692} C_VEL
LIN {X 0,Y 302.344,Z 977.53,A -85,B 0,C 180,E1 21672.486,E2 21672.486} C_VEL
LIN {X 0,Y 303.081,Z 977.53,A -85,B 0,C 180,E1 21681.36,E2 21681.36} C_VEL
LIN {X 0,Y 303.682,Z 977.53,A -85,B 0,C 180,E1 21687.127,E2 21687.127} C_VEL
LIN {X 0,Y 303.593,Z 977.53,A -85,B 0,C 180,E1 21693.183,E2 21693.183} C_VEL
LIN {X 0,Y 302.808,Z 977.53,A -85,B 0,C 180,E1 21701.533,E2 21701.533} C_VEL
LIN {X 0,Y 302.127,Z 977.53,A -85,B 0,C 180,E1 21710.539,E2 21710.539} C_VEL
LIN {X 0,Y 301.688,Z 977.53,A -85,B 0,C 180,E1 21716.859,E2 21716.859} C_VEL
LIN {X 0,Y 301.367,Z 977.53,A -85,B 0,C 180,E1 21723.562,E2 21723.562} C_VEL
LIN {X 0,Y 301.351,Z 977.53,A -85,B 0,C 180,E1 21728.92,E2 21728.92} C_VEL
LIN {X 0,Y 324.208,Z 1035.422,A -85,B 0,C 180,E1 21734.144,E2 21734.144} C_VEL
LIN {X 0,Y 337.244,Z 1076.181,A -85,B 0,C 180,E1 21738.068,E2 21738.068} C_VEL
LIN {X 0,Y 340.075,Z 1089.777,A -85,B 0,C 180,E1 21739.43,E2 21739.43} C_VEL
LIN {X 0,Y 332.411,Z 1127.928,A -85,B 0,C 180,E1 21742.768,E2 21742.768} C_VEL
LIN {X 0,Y 324.085,Z 1164.327,A -85,B 0,C 180,E1 21747.217,E2 21747.217} C_VEL
LIN {X 0,Y 316.448,Z 1195.662,A -85,B 0,C 180,E1 21752.536,E2 21752.536} C_VEL
LIN {X 0,Y 310.565,Z 1221.3,A -85,B 0,C 180,E1 21758.497,E2 21758.497} C_VEL
LIN {X 0,Y 306.764,Z 1240.982,A -85,B 0,C 180,E1 21764.829,E2 21764.829} C_VEL
LIN {X 0,Y 304.905,Z 1255.175,A -85,B 0,C 180,E1 21771.406,E2 21771.406} C_VEL
LIN {X 0,Y 304.337,Z 1263.206,A -85,B 0,C 180,E1 21777.126,E2 21777.126} C_VEL
LIN {X 0,Y 304.602,Z 1267.625,A -85,B 0,C 180,E1 21782.831,E2 21782.831} C_VEL
LIN {X 0,Y 305.77,Z 1268.844,A -85,B 0,C 180,E1 21788.528,E2 21788.528} C_VEL
LIN {X 0,Y 309.383,Z 1265.951,A -85,B 0,C 180,E1 21795.604,E2 21795.604} C_VEL
LIN {X 0,Y 318.456,Z 1256.437,A -85,B 0,C 180,E1 21803.832,E2 21803.832} C_VEL
LIN {X 0,Y 331.952,Z 1241.958,A -85,B 0,C 180,E1 21810.873,E2 21810.873} C_VEL
LIN {X 0,Y 352.549,Z 1220.113,A -85,B 0,C 180,E1 21817.741,E2 21817.741} C_VEL
LIN {X 0,Y 379.254,Z 1192.132,A -85,B 0,C 180,E1 21823.466,E2 21823.466} C_VEL
LIN {X 0,Y 380.694,Z 1190.66,A -85,B 0,C 180,E1 21823.71,E2 21823.71} C_VEL
LIN {X 0,Y 378.452,Z 1193.235,A -85,B 0,C 180,E1 21824.316,E2 21824.316} C_VEL
LIN {X 0,Y 353.191,Z 1222.565,A -85,B 0,C 180,E1 21829.253,E2 21829.253} C_VEL
LIN {X 0,Y 331.945,Z 1249.101,A -85,B 0,C 180,E1 21835.684,E2 21835.684} C_VEL
LIN {X 0,Y 316.154,Z 1271.267,A -85,B 0,C 180,E1 21843.697,E2 21843.697} C_VEL
LIN {X 0,Y 308.088,Z 1284.846,A -85,B 0,C 180,E1 21851.37,E2 21851.37} C_VEL
LIN {X 0,Y 304.962,Z 1292.176,A -85,B 0,C 180,E1 21858.55,E2 21858.55} C_VEL
LIN {X 0,Y 304.414,Z 1294.319,A -85,B 0,C 180,E1 21864.3,E2 21864.3} C_VEL
LIN {X 0,Y 304.836,Z 1293.011,A -85,B 0,C 180,E1 21870.013,E2 21870.013} C_VEL
LIN {X 0,Y 304.841,Z 1286.88,A -85,B 0,C 180,E1 21876.455,E2 21876.455} C_VEL
LIN {X 0,Y 305.443,Z 1275.427,A -85,B 0,C 180,E1 21882.913,E2 21882.913} C_VEL
LIN {X 0,Y 307.06,Z 1263.624,A -85,B 0,C 180,E1 21887.978,E2 21887.978} C_VEL
LIN {X 0,Y 312.386,Z 1248.712,A -85,B 0,C 180,E1 21895.129,E2 21895.129} C_VEL
LIN {X 0,Y 323.195,Z 1226.16,A -85,B 0,C 180,E1 21902.351,E2 21902.351} C_VEL
LIN {X 0,Y 337.977,Z 1197.842,A -85,B 0,C 180,E1 21908.52,E2 21908.52} C_VEL
LIN {X 0,Y 354.714,Z 1165.444,A -85,B 0,C 180,E1 21913.352,E2 21913.352} C_VEL
LIN {X 0,Y 371.038,Z 1130.797,A -85,B 0,C 180,E1 21916.901,E2 21916.901} C_VEL
LIN {X 0,Y 381.02,Z 1106.967,A -85,B 0,C 180,E1 21918.816,E2 21918.816} C_VEL
LIN {X 0,Y 381.502,Z 1096.211,A -85,B 0,C 180,E1 21921.485,E2 21921.485} C_VEL
LIN {X 0,Y 380.868,Z 1092.477,A -85,B 0,C 180,E1 21923.387,E2 21923.387} C_VEL
LIN {X 0,Y 379.699,Z 1090.644,A -85,B 0,C 180,E1 21926.954,E2 21926.954} C_VEL
LIN {X 0,Y 379.641,Z 1094.077,A -85,B 0,C 180,E1 21930.573,E2 21930.573} C_VEL
LIN {X 0,Y 379.592,Z 1102.014,A -85,B 0,C 180,E1 21933.469,E2 21933.469} C_VEL
LIN {X 0,Y 366.114,Z 1133.757,A -85,B 0,C 180,E1 21936.139,E2 21936.139} C_VEL
LIN {X 0,Y 362.87,Z 1140.446,A -85,B 0,C 180,E1 21936.869,E2 21936.869} C_VEL
LIN {X 0,Y 354.093,Z 1154.007,A -85,B 0,C 180,E1 21937.99,E2 21937.99} C_VEL
LIN {X 0,Y 345.909,Z 1165.01,A -85,B 0,C 180,E1 21939.087,E2 21939.087} C_VEL
LIN {X 0,Y 344.996,Z 1166.398,A -85,B 0,C 180,E1 21939.317,E2 21939.317} C_VEL
LIN {X 0,Y 330.266,Z 1187.623,A -85,B 0,C 180,E1 21944.043,E2 21944.043} C_VEL
LIN {X 0,Y 318.791,Z 1201.366,A -85,B 0,C 180,E1 21949.061,E2 21949.061} C_VEL
LIN {X 0,Y 310.058,Z 1209.619,A -85,B 0,C 180,E1 21954.412,E2 21954.412} C_VEL
LIN {X 0,Y 303.158,Z 1212.914,A -85,B 0,C 180,E1 21960.876,E2 21960.876} C_VEL
LIN {X 0,Y 299.63,Z 1209.817,A -85,B 0,C 180,E1 21967.283,E2 21967.283} C_VEL
LIN {X 0,Y 298.934,Z 1201.305,A -85,B 0,C 180,E1 21973.205,E2 21973.205} C_VEL
LIN {X 0,Y 300.085,Z 1186.421,A -85,B 0,C 180,E1 21979.18,E2 21979.18} C_VEL
LIN {X 0,Y 302.419,Z 1166.947,A -85,B 0,C 180,E1 21984.284,E2 21984.284} C_VEL
LIN {X 0,Y 306.039,Z 1142.586,A -85,B 0,C 180,E1 21988.682,E2 21988.682} C_VEL
LIN {X 0,Y 309.73,Z 1113.962,A -85,B 0,C 180,E1 21992.225,E2 21992.225} C_VEL
LIN {X 0,Y 312.935,Z 1082.773,A -85,B 0,C 180,E1 21994.697,E2 21994.697} C_VEL
LIN {X 0,Y 314.489,Z 1050.77,A -85,B 0,C 180,E1 21996.401,E2 21996.401} C_VEL
LIN {X 0,Y 298.551,Z 994.072,A -85,B 0,C 180,E1 22000.592,E2 22000.592} C_VEL
LIN {X 0,Y 293.363,Z 977.53,A -85,B 0,C 180,E1 22002.008,E2 22002.008} C_VEL
LIN {X 0,Y 293.078,Z 977.53,A -85,B 0,C 180,E1 22010.878,E2 22010.878} C_VEL
LIN {X 0,Y 293.464,Z 977.53,A -85,B 0,C 180,E1 22018.897,E2 22018.897} C_VEL
LIN {X 0,Y 293.944,Z 977.53,A -85,B 0,C 180,E1 22025.63,E2 22025.63} C_VEL
LIN {X 0,Y 294.4,Z 977.53,A -85,B 0,C 180,E1 22031.998,E2 22031.998} C_VEL
LIN {X 0,Y 294.856,Z 977.53,A -85,B 0,C 180,E1 22038.124,E2 22038.124} C_VEL
LIN {X 0,Y 295.771,Z 977.53,A -85,B 0,C 180,E1 22047.05,E2 22047.05} C_VEL
LIN {X 0,Y 295.771,Z 977.53,A -85,B 0,C 180,E1 22052.923,E2 22052.923} C_VEL
LIN {X 0,Y 294.838,Z 977.53,A -85,B 0,C 180,E1 22061.849,E2 22061.849} C_VEL
LIN {X 0,Y 294.365,Z 977.53,A -85,B 0,C 180,E1 22067.976,E2 22067.976} C_VEL
LIN {X 0,Y 293.911,Z 977.53,A -85,B 0,C 180,E1 22074.343,E2 22074.343} C_VEL
LIN {X 0,Y 293.531,Z 977.53,A -85,B 0,C 180,E1 22081.063,E2 22081.063} C_VEL
LIN {X 0,Y 293.417,Z 977.53,A -85,B 0,C 180,E1 22087.956,E2 22087.956} C_VEL
LIN {X 0,Y 316.081,Z 1034.677,A -85,B 0,C 180,E1 22093.307,E2 22093.307} C_VEL
LIN {X 0,Y 328.97,Z 1074.782,A -85,B 0,C 180,E1 22097.257,E2 22097.257} C_VEL
LIN {X 0,Y 332.64,Z 1091.207,A -85,B 0,C 180,E1 22098.973,E2 22098.973} C_VEL
LIN {X 0,Y 324.421,Z 1131.079,A -85,B 0,C 180,E1 22102.595,E2 22102.595} C_VEL
LIN {X 0,Y 315.993,Z 1166.709,A -85,B 0,C 180,E1 22107.148,E2 22107.148} C_VEL
LIN {X 0,Y 308.359,Z 1197.316,A -85,B 0,C 180,E1 22112.539,E2 22112.539} C_VEL
LIN {X 0,Y 302.335,Z 1223.437,A -85,B 0,C 180,E1 22118.873,E2 22118.873} C_VEL
LIN {X 0,Y 298.648,Z 1242.442,A -85,B 0,C 180,E1 22125.285,E2 22125.285} C_VEL
LIN {X 0,Y 296.897,Z 1256.083,A -85,B 0,C 180,E1 22131.912,E2 22131.912} C_VEL
LIN {X 0,Y 296.48,Z 1264.639,A -85,B 0,C 180,E1 22138.515,E2 22138.515} C_VEL
LIN {X 0,Y 297.119,Z 1268.995,A -85,B 0,C 180,E1 22145.833,E2 22145.833} C_VEL
LIN {X 0,Y 299.152,Z 1268.948,A -85,B 0,C 180,E1 22151.667,E2 22151.667} C_VEL
LIN {X 0,Y 305.821,Z 1263.281,A -85,B 0,C 180,E1 22160.27,E2 22160.27} C_VEL
LIN {X 0,Y 316.875,Z 1252.695,A -85,B 0,C 180,E1 22167.632,E2 22167.632} C_VEL
LIN {X 0,Y 335.429,Z 1234.755,A -85,B 0,C 180,E1 22175.14,E2 22175.14} C_VEL
LIN {X 0,Y 360.1,Z 1210.988,A -85,B 0,C 180,E1 22181.48,E2 22181.48} C_VEL
LIN {X 0,Y 372.194,Z 1199.478,A -85,B 0,C 180,E1 22183.767,E2 22183.767} C_VEL
LIN {X 0,Y 344.691,Z 1228.952,A -85,B 0,C 180,E1 22189.179,E2 22189.179} C_VEL
LIN {X 0,Y 323.397,Z 1253.625,A -85,B 0,C 180,E1 22195.803,E2 22195.803} C_VEL
LIN {X 0,Y 308.076,Z 1273.468,A -85,B 0,C 180,E1 22203.741,E2 22203.741} C_VEL
LIN {X 0,Y 299.5,Z 1286.846,A -85,B 0,C 180,E1 22212.343,E2 22212.343} C_VEL
LIN {X 0,Y 297.114,Z 1291.927,A -85,B 0,C 180,E1 22218.243,E2 22218.243} C_VEL
LIN {X 0,Y 296.516,Z 1293.827,A -85,B 0,C 180,E1 22224.148,E2 22224.148} C_VEL
LIN {X 0,Y 296.986,Z 1292.312,A -85,B 0,C 180,E1 22230.014,E2 22230.014} C_VEL
LIN {X 0,Y 297,Z 1285.853,A -85,B 0,C 180,E1 22236.626,E2 22236.626} C_VEL
LIN {X 0,Y 297.635,Z 1274.032,A -85,B 0,C 180,E1 22243.258,E2 22243.258} C_VEL
LIN {X 0,Y 299.004,Z 1264.234,A -85,B 0,C 180,E1 22247.716,E2 22247.716} C_VEL
LIN {X 0,Y 304.295,Z 1250.352,A -85,B 0,C 180,E1 22255.055,E2 22255.055} C_VEL
LIN {X 0,Y 315.026,Z 1229.319,A -85,B 0,C 180,E1 22262.388,E2 22262.388} C_VEL
LIN {X 0,Y 330.286,Z 1202.162,A -85,B 0,C 180,E1 22268.786,E2 22268.786} C_VEL
LIN {X 0,Y 347.589,Z 1171.135,A -85,B 0,C 180,E1 22273.781,E2 22273.781} C_VEL
LIN {X 0,Y 364.231,Z 1138.512,A -85,B 0,C 180,E1 22277.394,E2 22277.394} C_VEL
LIN {X 0,Y 376.698,Z 1111.168,A -85,B 0,C 180,E1 22279.613,E2 22279.613} C_VEL
LIN {X 0,Y 377.485,Z 1103.244,A -85,B 0,C 180,E1 22281.631,E2 22281.631} C_VEL
LIN {X 0,Y 377.134,Z 1099.428,A -85,B 0,C 180,E1 22283.49,E2 22283.49} C_VEL
LIN {X 0,Y 376.364,Z 1097.762,A -85,B 0,C 180,E1 22285.716,E2 22285.716} C_VEL
LIN {X 0,Y 375.871,Z 1099.484,A -85,B 0,C 180,E1 22289.374,E2 22289.374} C_VEL
LIN {X 0,Y 375.794,Z 1106.09,A -85,B 0,C 180,E1 22292.531,E2 22292.531} C_VEL
LIN {X 0,Y 361.569,Z 1137.113,A -85,B 0,C 180,E1 22295.245,E2 22295.245} C_VEL
LIN {X 0,Y 347.556,Z 1162.226,A -85,B 0,C 180,E1 22298.606,E2 22298.606} C_VEL
LIN {X 0,Y 344.996,Z 1166.398,A -85,B 0,C 180,E1 22299.317,E2 22299.317} C_VEL
LIN {X 0,Y 335.435,Z 1177.854,A -85,B 0,C 180,E1 22300.898,E2 22300.898} C_VEL
LIN {X 0,Y 326.722,Z 1186.825,A -85,B 0,C 180,E1 22302.414,E2 22302.414} C_VEL
LIN {X 0,Y 325.799,Z 1187.915,A -85,B 0,C 180,E1 22302.7,E2 22302.7} C_VEL
LIN {X 0,Y 312.593,Z 1202.758,A -85,B 0,C 180,E1 22308.133,E2 22308.133} C_VEL
LIN {X 0,Y 302.315,Z 1211.498,A -85,B 0,C 180,E1 22314.268,E2 22314.268} C_VEL
LIN {X 0,Y 295.991,Z 1214.082,A -85,B 0,C 180,E1 22320.021,E2 22320.021} C_VEL
LIN {X 0,Y 292.228,Z 1211.649,A -85,B 0,C 180,E1 22325.973,E2 22325.973} C_VEL
LIN {X 0,Y 291.034,Z 1203.925,A -85,B 0,C 180,E1 22332.041,E2 22332.041} C_VEL
LIN {X 0,Y 291.705,Z 1191.43,A -85,B 0,C 180,E1 22337.671,E2 22337.671} C_VEL
LIN {X 0,Y 293.785,Z 1173.324,A -85,B 0,C 180,E1 22343.058,E2 22343.058} C_VEL
LIN {X 0,Y 297.101,Z 1150.405,A -85,B 0,C 180,E1 22347.755,E2 22347.755} C_VEL
LIN {X 0,Y 301.029,Z 1121.978,A -85,B 0,C 180,E1 22351.734,E2 22351.734} C_VEL
LIN {X 0,Y 304.67,Z 1091.151,A -85,B 0,C 180,E1 22354.553,E2 22354.553} C_VEL
LIN {X 0,Y 306.946,Z 1051.958,A -85,B 0,C 180,E1 22356.823,E2 22356.823} C_VEL
LIN {X 0,Y 291.416,Z 996.641,A -85,B 0,C 180,E1 22361.042,E2 22361.042} C_VEL
LIN {X 0,Y 285.366,Z 977.53,A -85,B 0,C 180,E1 22362.665,E2 22362.665} C_VEL
LIN {X 0,Y 285.106,Z 977.53,A -85,B 0,C 180,E1 22370.356,E2 22370.356} C_VEL
LIN {X 0,Y 285.466,Z 977.53,A -85,B 0,C 180,E1 22378.164,E2 22378.164} C_VEL
LIN {X 0,Y 285.892,Z 977.53,A -85,B 0,C 180,E1 22384.896,E2 22384.896} C_VEL
LIN {X 0,Y 286.498,Z 977.53,A -85,B 0,C 180,E1 22392.226,E2 22392.226} C_VEL
LIN {X 0,Y 287.176,Z 977.53,A -85,B 0,C 180,E1 22400.878,E2 22400.878} C_VEL
LIN {X 0,Y 288.005,Z 977.53,A -85,B 0,C 180,E1 22409.155,E2 22409.155} C_VEL
LIN {X 0,Y 287.504,Z 977.53,A -85,B 0,C 180,E1 22416.037,E2 22416.037} C_VEL
LIN {X 0,Y 286.903,Z 977.53,A -85,B 0,C 180,E1 22422.182,E2 22422.182} C_VEL
LIN {X 0,Y 286.365,Z 977.53,A -85,B 0,C 180,E1 22428.496,E2 22428.496} C_VEL
LIN {X 0,Y 285.788,Z 977.53,A -85,B 0,C 180,E1 22435.628,E2 22435.628} C_VEL
LIN {X 0,Y 285.493,Z 977.53,A -85,B 0,C 180,E1 22442.04,E2 22442.04} C_VEL
LIN {X 0,Y 285.448,Z 977.53,A -85,B 0,C 180,E1 22446.922,E2 22446.922} C_VEL
LIN {X 0,Y 308.404,Z 1035.247,A -85,B 0,C 180,E1 22452.561,E2 22452.561} C_VEL
LIN {X 0,Y 321.182,Z 1075.145,A -85,B 0,C 180,E1 22456.615,E2 22456.615} C_VEL
LIN {X 0,Y 325.28,Z 1092.224,A -85,B 0,C 180,E1 22458.469,E2 22458.469} C_VEL
LIN {X 0,Y 317.148,Z 1130.764,A -85,B 0,C 180,E1 22462.044,E2 22462.044} C_VEL
LIN {X 0,Y 308.248,Z 1167.593,A -85,B 0,C 180,E1 22466.854,E2 22466.854} C_VEL
LIN {X 0,Y 300.774,Z 1196.954,A -85,B 0,C 180,E1 22472.136,E2 22472.136} C_VEL
LIN {X 0,Y 294.673,Z 1222.748,A -85,B 0,C 180,E1 22478.473,E2 22478.473} C_VEL
LIN {X 0,Y 290.601,Z 1243.513,A -85,B 0,C 180,E1 22485.64,E2 22485.64} C_VEL
